(* IEC 61131-3 sources: cc_kush_rewrite/POUs, 10 files *)

(* ---- GLOBAL.st ---- *)
VAR_GLOBAL
	// Системные ФБ
	PULSE : BLINK;
	PULSE_RTRIG : R_TRIG;

	// Системные флаги
	xStateEmergencyStop : BOOL; // Система была аварийно остановлена
	xStateErrorAcceptIdle : BOOL; // Невозможно принять коэффицент шихтования по заданию оператора - сумма коэффицентов не равна 100
	xStateErrorCheckReady : BOOL; // Проверки стадии готовности к пуску провалились
	xStateAutoWorking : BOOL; // Система полностью запущена и работает в автоматическом режиме
	// Расчёт КИУМ
	ICUR_PRECENT : REAL; // Коэффициент использования установленной мощности (в процентах)
	rElectricityMeter : REAL; // Раход электроэнергии

	// Ограничение производительности
	EFFICIENCY_LIMIT_RATE : REAL := 1; // Коэффицент ограничения производительности (0-1)

	// Переменные симуляции
	SIMULATION : BOOL := FALSE;
	SIMULATION_BUNKER_WEIGHT : BOOL := FALSE; // Включение симуляции расхода и пополнения веса бункеров

	// == MODBUS РЕГИСТРЫ ДЛЯ SCADA ==
	// Массив регистров для передачи данных в SCADA систему
	awModbusInputRegisters : ARRAY [0..511] OF WORD; // Modbus Input регистры
	awModbusHoldingRegisters : ARRAY [0..511] OF WORD; // Modbus Holding регистры

	// == СИГНАЛЫ СВЯЗИ СО SCADA ==
	SCADA_HEARTBEAT : BOOL := FALSE; // Пульсирующий сигнал от SCADA (0 → 1 → 0) для контроля связи

END_VAR
VAR_GLOBAL RETAIN
	// == КРИТИЧЕСКИЕ НАСТРОЙКИ ==
	DISABLE_AUTO_STOPPING : BOOL := FALSE; // Отключение автоматических блокировок по цепям безопасности механизмов
	DISABLE_AUTO_STOPPING_DEPENDENCIES : BOOL := FALSE; 			// Отключение автоматических блокировок по блокировочным зависимостям
	DISABLE_AUTO_STOPPING_DEPENDENCIES_BUNKER1 : BOOL := FALSE; 	// Отключение автоматических блокировок бункера 1
	DISABLE_AUTO_STOPPING_DEPENDENCIES_BUNKER2 : BOOL := FALSE; 	// Отключение автоматических блокировок бункера 2
	DISABLE_AUTO_STOPPING_DEPENDENCIES_BUNKER3 : BOOL := FALSE; 	// Отключение автоматических блокировок бункера 3
	DISABLE_AUTO_STOPPING_DEPENDENCIES_CONVEYOR : BOOL := FALSE; 	// Отключение автоматических блокировок сборного конвейера
	DISABLE_AUTO_STOPPING_DEPENDENCIES_DUMPER : BOOL := FALSE; 		// Отключение автоматических блокировок отвалообразователя

	DISABLE_AUTO_STOPPING_SCADA_COMMUNICATION : BOOL := TRUE; // Отключение автоматических блокировок по потере связи со SCADA
	DISABLE_AUTO_STOPPING_CURRENT : BOOL := FALSE; // Отключение автоматических блокировок по значению тока
	BUNKER_INSTANT_STOP : BOOL := FALSE; // Флаг мгновенной остановки бункеров (TRUE = одновременная остановка всех 3-х бункеров, FALSE = последовательная остановка)

	// == УСТАВКИ ==
	VFD_FREQUENCY_MAX : REAL := 50;
	VFD_FREQUENCY_STEP : REAL := 2;
	VFD_FREQUENCY_INACCURANCY : REAL := 0.5;
	VFD_FREQUENCY_SYNC_TOLERANCE : REAL := 1.5; // Допустимая разница частот для синхронизации моторов

		// == ПАРАМЕТРЫ АЦП/ЦАП ДЛЯ ЧРП ==
	VFD_ADC_MAX : INT := 27648; // Максимальный код АЦП (аналоговый вход/выход)
	VFD_ADC_MIN : INT := 0; // Минимальный код АЦП
	VFD_FREQ_MIN : REAL := 0.0; // Минимальная частота ЧРП (Гц)
	VFD_FREQ_MAX_RANGE : REAL := 50.0; // Максимальная частота для масштабирования АЦП (Гц)

	// == ПАРАМЕТРЫ ТОКА 4-20 мА ==
	VFD_CURRENT_MIN : REAL := 4.0; // Минимальный ток (мА)
	VFD_CURRENT_MAX : REAL := 20.0; // Максимальный ток (мА)
	VFD_CURRENT_ALARM_LL : REAL := 3.8; // Аварийно низкий уровень тока (обрыв линии)
	VFD_CURRENT_ALARM_L : REAL := 4.5; // Низкий уровень тока
	VFD_CURRENT_ALARM_H : REAL := 19.5; // Высокий уровень тока
	VFD_CURRENT_ALARM_HH : REAL := 20.2; // Аварийно высокий уровень тока (перегрузка)

	// == ПАРАМЕТРЫ ДИАПАЗОНА ТЕМПЕРАТУР ==
	TEMP_BEARING_MIN : REAL := 0.0; // Минимальная температура подшипникового узла (°C)
	TEMP_BEARING_MAX : REAL := 100.0; // Максимальная температура подшипникового узла (°C)

	// Настройка виброобрушения
	VIBRATOR_SETTINGS : ST_BunkerVibratorSettings := (
		TIME_ACTIVE := T#15S,
		TIME_PAUSE_VIBRATOR := T#30S,
		TIME_PAUSE_FB := T#30S,
		COUNT_CYCLE := 3
		);

	// Настройка пневмообрушения
	PNEUMO_SETTINGS : ST_BunkerVibratorSettings := (
		TIME_ACTIVE := T#10S,
		TIME_PAUSE_VIBRATOR := T#10S,
		TIME_PAUSE_FB := T#30S,
		COUNT_CYCLE := 3
		);

	// Опция плавного задания частоты
	VFD_SMOOTH_SET_FREQUENCY : BOOL := FALSE;

	// Таймеры последовательного запуска механизмов в автоматическом режиме
	TIME_AFTER_START_DUMPER : TIME := T#120S; // Время ожидания после запуска отвалообразователя
	TIME_AFTER_START_CONVEYOR : TIME := T#120S; // Время ожидания после запуска конвейера
	TIME_AFTER_START_BUNKER_1 : TIME := T#120S; // Время ожидания после запуска бункера 1
	TIME_AFTER_START_BUNKER_2 : TIME := T#120S; // Время ожидания после запуска бункера 2
	TIME_AFTER_START_BUNKER_3 : TIME := T#120S; // Время ожидания после запуска бункера 3

	// Таймеры контроля выполнения команд (тайм-ауты)
	TIME_TIMEOUT_STOP_DUMPER : TIME := T#30S; // Тайм-аут остановки отвалообразователя (WORK → IDLE)
	TIME_TIMEOUT_STOP_CONVEYOR : TIME := T#30S; // Тайм-аут остановки конвейера (WORK → IDLE)
	TIME_TIMEOUT_ROTATION_DUMPER : TIME := T#20S; // Тайм-аут выполнения команд поворота дампера
	TIME_TIMEOUT_STOP_BUNKER : TIME := T#20S; // Тайм-аут остановки вибропитателей бункера (WORK → IDLE)

	// Таймер ожидания пропавшего сигнала обратной связи работы механизма
	TIME_WAITING_FEEDBACK : TIME := T#0S;

	// == ПАРАМЕТРЫ СВЯЗИ СО SCADA ==
	SCADA_HEARTBEAT_TIMEOUT : TIME := T#5S; // Таймаут отсутствия изменений heartbeat сигнала (потеря связи)

	// Таймаут контроля суммы пропорций в режиме WORK
	BUNKER_PROPORTION_SUM_TIMEOUT : TIME := T#20S; // Время ожидания корректировки суммы пропорций оператором (сумма должна быть = 100%)

	// Скорость конвейера
	CONVEYOR_DEAFULT_SPEED : REAL := -1;

	// Температура подшипникового узла мотора вибропитателя
	MOTOR_VIBFEEDER_TEMP_POINTS : ST_AlarmSetpoints := (
		LL_Value := -1,
		L_Value := -1,
		H_Value := -1,
		HH_Value := -1);
	// Ток мотора вибропитателя
	MOTOR_VIBFEEDER_CURRENT_POINTS : ST_AlarmSetpoints := (
		LL_Value := -1,
		L_Value := -1,
		H_Value := -1,
		HH_Value := -1);
	// Ток мотора вибратора
	MOTOR_VIBRATOR_CURRENT_POINTS : ST_AlarmSetpoints := (
		LL_Value := -1,
		L_Value := -1,
		H_Value := -1,
		HH_Value := -1);
	// Ток мотора конвейера отвалообразователя
	MOTOR_CONVEYOR_CURRENT_POINTS : ST_AlarmSetpoints := (
		LL_Value := -1,
		L_Value := -1,
		H_Value := -1,
		HH_Value := -1);
	// Ток мотора конвейера сборного
	MOTOR_CONVEYOR_PREFABRICATED_CURRENT_POINTS : ST_AlarmSetpoints := (
		LL_Value := -1,
		L_Value := -1,
		H_Value := -1,
		HH_Value := -1);
	// Ток мотора поворота отвалообразователя
	MOTOR_ROTATION_CURRENT_POINTS : ST_AlarmSetpoints := (
		LL_Value := -1,
		L_Value := -1,
		H_Value := -1,
		HH_Value := -1);

	// Предпусковая сигнализация конвейера отвалообразователя
	DUMPER_CONVEYOR_PRESTART_ALARM_SETTINGS : ST_PreStartAlarmSettings := (
		OPTION_ENABLE := TRUE, // Опция на включение ППЗ в алгоритм
		TIME_FIRST_SIGNAL := T#3S, // Время звучания первого сигнала
		TIME_FIRST_SIGNAL_PAUSE := T#3S, // Пауза после первого сигнала
		TIME_SECOND_SIGNAL := T#3S, // Время звучания второго сигнала
		TIME_SECOND_SIGNAL_PAUSE := T#3S); // Пауза после втотрого сигнала

	// Предпусковая сигнализация сборного конвейера
	CONVEYOR_PRESTART_ALARM_SETTINGS : ST_PreStartAlarmSettings := (
		OPTION_ENABLE := TRUE, // Опция на включение ППЗ в алгоритм
		TIME_FIRST_SIGNAL := T#3S, // Время звучания первого сигнала
		TIME_FIRST_SIGNAL_PAUSE := T#3S, // Пауза после первого сигнала
		TIME_SECOND_SIGNAL := T#3S, // Время звучания второго сигнала
		TIME_SECOND_SIGNAL_PAUSE := T#3S); // Пауза после втотрого сигнала

	// Световая индикация Гц
	ANNUNCIATOR_LIGHT_HZ : REAL := 2;

	// Частота мотора конвейера
	MOTOR_FREQUENCY_CONVEYOR : REAL := 50;
	// Частота мотора конвейера отвалообразователя
	MOTOR_FREQUENCY_DUMPER_CONVEYOR : REAL := 50;
	// Частота мотора поворота отвалообразователя
	MOTOR_FREQUENCY_DUMPER_ROTATION : REAL := -1;

	BUNKER_MINIMAL_WEIGHT :REAL := 0; // Уставка минимального веса бункера. Результат <= считывается алгоритмом как пустой бункер.

	// Уставки бункера
	PNEUMATIC_COLLAPSE_TIME : TIME := T#0S; // Уставка времени таймера пневмообрушения
	BUNKER_WORK_PRECENT_1 : REAL; // Уставка пропорции шихтования для бункера 1
	BUNKER_WORK_PRECENT_2 : REAL; // Уставка пропорции шихтования для бункера 2
	BUNKER_WORK_PRECENT_3 : REAL; // Уставка пропорции шихтования для бункера 3
	BUNKER_VIBFEEDER_START_FREQUENCY : REAL := 10.0; // Минимальная частота для запуска вибропитателей (Гц)
	BUNKER_VIBFEEDER_FREQUENCY_TARGET_SUM : REAL := 50.0; // Целевая суммарная частота вибропитателей (Гц)
    BUNKER_ENABLE_PID : BOOL := FALSE;
    BUNKER_ENABLE_PROPORTION_MONITORING : BOOL := FALSE;

	// == КОНТРОЛЬ МИНИМАЛЬНОЙ И МАКСИМАЛЬНОЙ ЧАСТОТЫ ВИБРОПИТАТЕЛЯ (ДЛЯ ПИД-РЕГУЛЯТОРА) ==
	BUNKER_VIBFEEDER_MIN_FREQUENCY_LIMIT : REAL := 5.0; // Минимальная допустимая частота вибропитателя (Гц) - при достижении этой уставки запускается таймер аварии
	BUNKER_VIBFEEDER_MIN_FREQUENCY_TIMEOUT : TIME := T#30S; // Время задержки перед аварийной остановкой при достижении минимальной частоты
	BUNKER_VIBFEEDER_MAX_FREQUENCY_LIMIT : REAL := 50.0; // Максимальная допустимая частота вибропитателя (Гц) - при достижении этой уставки запускается таймер аварии
	BUNKER_VIBFEEDER_MAX_FREQUENCY_TIMEOUT : TIME := T#30S; // Время задержки перед аварийной остановкой при достижении максимальной частоты

	// Ручное задание частоты на бункер (работает в ручном режиме управления)
	BUNKER_1_FREQ_VIBFEEDER : REAL := 30;
	BUNKER_1_FREQ_VIBRATOR : REAL := 30;
	BUNKER_2_FREQ_VIBFEEDER : REAL := 30;
	BUNKER_2_FREQ_VIBRATOR : REAL := 30;
	BUNKER_3_FREQ_VIBFEEDER : REAL := 30;
	BUNKER_3_FREQ_VIBRATOR : REAL := 30;

	// Светофор бункера
	BUNKER_WEIGHT_LIGHT_RED : REAL := 90; // Уставка веса бункера для красного светофора
	BUNKER_WEIGHT_LIGHT_YELLOW : REAL := 80; // Уставка веса бункера для жёлтого светофора
	BUNKER_WEIGHT_LIGHT_GREEN : REAL := 50; // Уставка веса бункера для зелёного светофора

	BUNKER_WEIGHT_LIGHT_RED_SPECIAL : REAL := 10; // Уставка веса бункера для красного светофора, когда сырье закончилось и требуется остановить подачу материала в остальные бункеры для будущего алгоритма опустошения

	// Константы
	AMOUNT_BUNKER_MOTOR_VIBFEEDER : INT := 2;
	AMOUNT_BUNKER_MOTOR_VIBRATOR : INT := 4;
END_VAR

(* ---- FC_ModbusToSCADA.st ---- *)
FUNCTION FC_ModbusToSCADA : BOOL
VAR_INPUT
    stBunker : REFERENCE TO ARRAY [1..3] OF ST_Bunker;
    stDumper : REFERENCE TO ST_DUMPER;
    stConveyor : REFERENCE TO ST_ConveyorPrefabricated;
    stCommonSignals : REFERENCE TO ST_CommonSignals;
	stCommands : REFERENCE TO ST_Commands;
	eBunkerStageToSCADA : REFERENCE TO ARRAY[1..3] OF E_ScadaStatesDevice;
	eConveyorStageToSCADA : REFERENCE TO E_ScadaStatesDevice; // Состояние для SCADA конвейера
	eDumperStageToSCADA : REFERENCE TO E_ScadaStatesDevice; // Состояние для SCADA отвалообразователя
	eSystemStageToSCADA : REFERENCE TO E_ScadaStatesDevice; // Общее состояние системы для SCADA
	fbScadaCommunication : REFERENCE TO FB_ScadaCommunication; // Функциональный блок контроля связи со SCADA

END_VAR
VAR
	rTempTime : REAL;
END_VAR

// ========================================
// MODBUS РЕГИСТРЫ
// ========================================

// === HOLDING РЕГИСТРЫ (SCADA → PLC) - Чтение уставок ===

// Общие системные переменные и уставки (0-29)
// Регистры 0-1: BOOL флаги команд
FC_ModbusReadBool(pRegisters := ADR(awModbusHoldingRegisters), iRegisterIndex := 0, iBitIndex := 0, xValue => stCommands.cmdStartCommon.ixSignal);
FC_ModbusReadBool(pRegisters := ADR(awModbusHoldingRegisters), iRegisterIndex := 0, iBitIndex := 1, xValue => stCommands.cmdStopCommon.ixSignal);
FC_ModbusReadBool(pRegisters := ADR(awModbusHoldingRegisters), iRegisterIndex := 0, iBitIndex := 2, xValue => stCommands.cmdEmergencyStopCommon.ixSignal);
FC_ModbusReadBool(pRegisters := ADR(awModbusHoldingRegisters), iRegisterIndex := 0, iBitIndex := 3, xValue => stCommands.cmdResetAll.ixSignal);
FC_ModbusReadBool(pRegisters := ADR(awModbusHoldingRegisters), iRegisterIndex := 0, iBitIndex := 4, xValue => SCADA_HEARTBEAT);
//FC_ModbusReadBool(pRegisters := ADR(awModbusHoldingRegisters), iRegisterIndex := 0, iBitIndex := 5, xValue => DISABLE_AUTO_STOPPING_SCADA_COMMUNICATION);
FC_ModbusReadBool(pRegisters := ADR(awModbusHoldingRegisters), iRegisterIndex := 0, iBitIndex := 8, xValue => stCommands.cmdSetToRepair);
FC_ModbusReadBool(pRegisters := ADR(awModbusHoldingRegisters), iRegisterIndex := 0, iBitIndex := 9, xValue => stCommands.cmdSetToManual);
FC_ModbusReadBool(pRegisters := ADR(awModbusHoldingRegisters), iRegisterIndex := 0, iBitIndex := 10, xValue => stCommands.cmdSetToAuto);

// Уставки ЧРП (30-59)
// Регистры 30-31: BOOL флаги ЧРП
FC_ModbusReadBool(pRegisters := ADR(awModbusHoldingRegisters), iRegisterIndex := 30, iBitIndex := 0, xValue => VFD_SMOOTH_SET_FREQUENCY);

FC_ModbusReadReal(pRegisters := ADR(awModbusHoldingRegisters), iRegisterIndex := 32, rValue => VFD_FREQUENCY_MAX);
FC_ModbusReadReal(pRegisters := ADR(awModbusHoldingRegisters), iRegisterIndex := 34, rValue => VFD_FREQUENCY_STEP);
FC_ModbusReadReal(pRegisters := ADR(awModbusHoldingRegisters), iRegisterIndex := 36, rValue => VFD_FREQUENCY_INACCURANCY);
FC_ModbusReadReal(pRegisters := ADR(awModbusHoldingRegisters), iRegisterIndex := 38, rValue => VFD_FREQUENCY_SYNC_TOLERANCE);
FC_ModbusReadReal(pRegisters := ADR(awModbusHoldingRegisters), iRegisterIndex := 40, rValue => MOTOR_FREQUENCY_CONVEYOR);
FC_ModbusReadReal(pRegisters := ADR(awModbusHoldingRegisters), iRegisterIndex := 42, rValue => MOTOR_FREQUENCY_DUMPER_CONVEYOR);
FC_ModbusReadReal(pRegisters := ADR(awModbusHoldingRegisters), iRegisterIndex := 44, rValue => MOTOR_FREQUENCY_DUMPER_ROTATION);
FC_ModbusReadReal(pRegisters := ADR(awModbusHoldingRegisters), iRegisterIndex := 46, rValue => CONVEYOR_DEAFULT_SPEED);

// Уставки бункеров (60-89)
// Регистры 60-61: BOOL флаги (резерв)
FC_ModbusReadReal(pRegisters := ADR(awModbusHoldingRegisters), iRegisterIndex := 62, rValue => BUNKER_WORK_PRECENT_1);
FC_ModbusReadReal(pRegisters := ADR(awModbusHoldingRegisters), iRegisterIndex := 64, rValue => BUNKER_WORK_PRECENT_2);
FC_ModbusReadReal(pRegisters := ADR(awModbusHoldingRegisters), iRegisterIndex := 66, rValue => BUNKER_WORK_PRECENT_3);
FC_ModbusReadReal(pRegisters := ADR(awModbusHoldingRegisters), iRegisterIndex := 68, rValue => BUNKER_MINIMAL_WEIGHT);
FC_ModbusReadReal(pRegisters := ADR(awModbusHoldingRegisters), iRegisterIndex := 70, rValue => BUNKER_WEIGHT_LIGHT_RED_SPECIAL);
FC_ModbusReadReal(pRegisters := ADR(awModbusHoldingRegisters), iRegisterIndex := 72, rValue => BUNKER_WEIGHT_LIGHT_RED);
FC_ModbusReadReal(pRegisters := ADR(awModbusHoldingRegisters), iRegisterIndex := 74, rValue => BUNKER_WEIGHT_LIGHT_YELLOW);
FC_ModbusReadReal(pRegisters := ADR(awModbusHoldingRegisters), iRegisterIndex := 76, rValue => BUNKER_WEIGHT_LIGHT_GREEN);

// Уставки аварийных значений - Температура (90-119)
// Регистры 90-91: BOOL флаги (резерв)
FC_ModbusReadReal(pRegisters := ADR(awModbusHoldingRegisters), iRegisterIndex := 92, rValue => MOTOR_VIBFEEDER_TEMP_POINTS.LL_Value);
FC_ModbusReadReal(pRegisters := ADR(awModbusHoldingRegisters), iRegisterIndex := 94, rValue => MOTOR_VIBFEEDER_TEMP_POINTS.L_Value);
FC_ModbusReadReal(pRegisters := ADR(awModbusHoldingRegisters), iRegisterIndex := 96, rValue => MOTOR_VIBFEEDER_TEMP_POINTS.H_Value);
FC_ModbusReadReal(pRegisters := ADR(awModbusHoldingRegisters), iRegisterIndex := 98, rValue => MOTOR_VIBFEEDER_TEMP_POINTS.HH_Value);

// Уставки аварийных значений - Ток (120-149)
// Регистры 120-121: BOOL флаги (резерв)
FC_ModbusReadReal(pRegisters := ADR(awModbusHoldingRegisters), iRegisterIndex := 122, rValue => MOTOR_VIBFEEDER_CURRENT_POINTS.LL_Value);
FC_ModbusReadReal(pRegisters := ADR(awModbusHoldingRegisters), iRegisterIndex := 124, rValue => MOTOR_VIBFEEDER_CURRENT_POINTS.L_Value);
FC_ModbusReadReal(pRegisters := ADR(awModbusHoldingRegisters), iRegisterIndex := 126, rValue => MOTOR_VIBFEEDER_CURRENT_POINTS.H_Value);
FC_ModbusReadReal(pRegisters := ADR(awModbusHoldingRegisters), iRegisterIndex := 128, rValue => MOTOR_VIBFEEDER_CURRENT_POINTS.HH_Value);
FC_ModbusReadReal(pRegisters := ADR(awModbusHoldingRegisters), iRegisterIndex := 130, rValue => MOTOR_VIBRATOR_CURRENT_POINTS.LL_Value);
FC_ModbusReadReal(pRegisters := ADR(awModbusHoldingRegisters), iRegisterIndex := 132, rValue => MOTOR_VIBRATOR_CURRENT_POINTS.L_Value);
FC_ModbusReadReal(pRegisters := ADR(awModbusHoldingRegisters), iRegisterIndex := 134, rValue => MOTOR_VIBRATOR_CURRENT_POINTS.H_Value);
FC_ModbusReadReal(pRegisters := ADR(awModbusHoldingRegisters), iRegisterIndex := 136, rValue => MOTOR_VIBRATOR_CURRENT_POINTS.HH_Value);
FC_ModbusReadReal(pRegisters := ADR(awModbusHoldingRegisters), iRegisterIndex := 138, rValue => MOTOR_CONVEYOR_CURRENT_POINTS.LL_Value);
FC_ModbusReadReal(pRegisters := ADR(awModbusHoldingRegisters), iRegisterIndex := 140, rValue => MOTOR_CONVEYOR_CURRENT_POINTS.L_Value);
FC_ModbusReadReal(pRegisters := ADR(awModbusHoldingRegisters), iRegisterIndex := 142, rValue => MOTOR_CONVEYOR_CURRENT_POINTS.H_Value);
FC_ModbusReadReal(pRegisters := ADR(awModbusHoldingRegisters), iRegisterIndex := 144, rValue => MOTOR_CONVEYOR_CURRENT_POINTS.HH_Value);
FC_ModbusReadReal(pRegisters := ADR(awModbusHoldingRegisters), iRegisterIndex := 146, rValue => MOTOR_ROTATION_CURRENT_POINTS.LL_Value);
FC_ModbusReadReal(pRegisters := ADR(awModbusHoldingRegisters), iRegisterIndex := 148, rValue => MOTOR_ROTATION_CURRENT_POINTS.L_Value);

// Уставки времени (150-179)
// Регистры 150-151: Уставки связи со SCADA
FC_ModbusReadReal(pRegisters := ADR(awModbusHoldingRegisters), iRegisterIndex := 150, rValue => rTempTime);
SCADA_HEARTBEAT_TIMEOUT := REAL_TO_TIME(rTempTime * 1000); // Таймаут потери связи (секунды)

FC_ModbusReadReal(pRegisters := ADR(awModbusHoldingRegisters), iRegisterIndex := 152, rValue => MOTOR_ROTATION_CURRENT_POINTS.H_Value);
FC_ModbusReadReal(pRegisters := ADR(awModbusHoldingRegisters), iRegisterIndex := 154, rValue => MOTOR_ROTATION_CURRENT_POINTS.HH_Value);
FC_ModbusReadReal(pRegisters := ADR(awModbusHoldingRegisters), iRegisterIndex := 156, rValue => rTempTime);
//VIBRATOR_SETTINGS.TIME_ACTIVE := REAL_TO_TIME(rTempTime * 1000);
FC_ModbusReadReal(pRegisters := ADR(awModbusHoldingRegisters), iRegisterIndex := 158, rValue => rTempTime);
//VIBRATOR_SETTINGS.TIME_PAUSE_VIBRATOR := REAL_TO_TIME(rTempTime * 1000);
FC_ModbusReadReal(pRegisters := ADR(awModbusHoldingRegisters), iRegisterIndex := 160, rValue => rTempTime);
VIBRATOR_SETTINGS.TIME_PAUSE_FB := REAL_TO_TIME(rTempTime * 1000);
FC_ModbusReadReal(pRegisters := ADR(awModbusHoldingRegisters), iRegisterIndex := 162, rValue => rTempTime);
PNEUMO_SETTINGS.TIME_ACTIVE := REAL_TO_TIME(rTempTime * 1000);
FC_ModbusReadReal(pRegisters := ADR(awModbusHoldingRegisters), iRegisterIndex := 164, rValue => rTempTime);
PNEUMO_SETTINGS.TIME_PAUSE_VIBRATOR := REAL_TO_TIME(rTempTime * 1000);
FC_ModbusReadReal(pRegisters := ADR(awModbusHoldingRegisters), iRegisterIndex := 166, rValue => rTempTime);
PNEUMO_SETTINGS.TIME_PAUSE_FB := REAL_TO_TIME(rTempTime * 1000);
FC_ModbusReadReal(pRegisters := ADR(awModbusHoldingRegisters), iRegisterIndex := 168, rValue => rTempTime);
TIME_WAITING_FEEDBACK := REAL_TO_TIME(rTempTime * 1000);
FC_ModbusReadReal(pRegisters := ADR(awModbusHoldingRegisters), iRegisterIndex := 170, rValue => rTempTime);
PNEUMATIC_COLLAPSE_TIME := REAL_TO_TIME(rTempTime * 1000);
FC_ModbusReadReal(pRegisters := ADR(awModbusHoldingRegisters), iRegisterIndex := 172, rValue => rTempTime);
DUMPER_CONVEYOR_PRESTART_ALARM_SETTINGS.TIME_FIRST_SIGNAL := REAL_TO_TIME(rTempTime * 1000);
FC_ModbusReadReal(pRegisters := ADR(awModbusHoldingRegisters), iRegisterIndex := 174, rValue => rTempTime);
DUMPER_CONVEYOR_PRESTART_ALARM_SETTINGS.TIME_FIRST_SIGNAL_PAUSE := REAL_TO_TIME(rTempTime * 1000);
FC_ModbusReadReal(pRegisters := ADR(awModbusHoldingRegisters), iRegisterIndex := 176, rValue => rTempTime);
DUMPER_CONVEYOR_PRESTART_ALARM_SETTINGS.TIME_SECOND_SIGNAL := REAL_TO_TIME(rTempTime * 1000);
FC_ModbusReadReal(pRegisters := ADR(awModbusHoldingRegisters), iRegisterIndex := 178, rValue => rTempTime);
DUMPER_CONVEYOR_PRESTART_ALARM_SETTINGS.TIME_SECOND_SIGNAL_PAUSE := REAL_TO_TIME(rTempTime * 1000);

// Уставки времени (продолжение) (180-209)
// Регистры 180-181: BOOL флаги (резерв)
FC_ModbusReadReal(pRegisters := ADR(awModbusHoldingRegisters), iRegisterIndex := 182, rValue => rTempTime);
CONVEYOR_PRESTART_ALARM_SETTINGS.TIME_FIRST_SIGNAL := REAL_TO_TIME(rTempTime * 1000);
FC_ModbusReadReal(pRegisters := ADR(awModbusHoldingRegisters), iRegisterIndex := 184, rValue => rTempTime);
CONVEYOR_PRESTART_ALARM_SETTINGS.TIME_FIRST_SIGNAL_PAUSE := REAL_TO_TIME(rTempTime * 1000);
FC_ModbusReadReal(pRegisters := ADR(awModbusHoldingRegisters), iRegisterIndex := 186, rValue => rTempTime);
CONVEYOR_PRESTART_ALARM_SETTINGS.TIME_SECOND_SIGNAL := REAL_TO_TIME(rTempTime * 1000);
FC_ModbusReadReal(pRegisters := ADR(awModbusHoldingRegisters), iRegisterIndex := 188, rValue => rTempTime);
CONVEYOR_PRESTART_ALARM_SETTINGS.TIME_SECOND_SIGNAL_PAUSE := REAL_TO_TIME(rTempTime * 1000);

// Команды - Отвалообразователь (210-239)
// Регистры 210-211: BOOL флаги управления отвалообразователем
FC_ModbusReadBool(pRegisters := ADR(awModbusHoldingRegisters), iRegisterIndex := 210, iBitIndex := 0, xValue => stDumper.cmdStartConveyor);
FC_ModbusReadBool(pRegisters := ADR(awModbusHoldingRegisters), iRegisterIndex := 210, iBitIndex := 1, xValue => stDumper.cmdStopConveyor);
FC_ModbusReadBool(pRegisters := ADR(awModbusHoldingRegisters), iRegisterIndex := 210, iBitIndex := 2, xValue => stDumper.cmdEmergencyStop);
FC_ModbusReadBool(pRegisters := ADR(awModbusHoldingRegisters), iRegisterIndex := 210, iBitIndex := 3, xValue => stDumper.cmdReset);
FC_ModbusReadBool(pRegisters := ADR(awModbusHoldingRegisters), iRegisterIndex := 210, iBitIndex := 8, xValue => stDumper.cmdSetModeRepair);
FC_ModbusReadBool(pRegisters := ADR(awModbusHoldingRegisters), iRegisterIndex := 210, iBitIndex := 9, xValue => stDumper.cmdSetModeManual);
FC_ModbusReadBool(pRegisters := ADR(awModbusHoldingRegisters), iRegisterIndex := 210, iBitIndex := 10, xValue => stDumper.cmdSetModeAuto);
FC_ModbusReadBool(pRegisters := ADR(awModbusHoldingRegisters), iRegisterIndex := 210, iBitIndex := 11, xValue => stDumper.cmdBuildCircuitOn);
FC_ModbusReadBool(pRegisters := ADR(awModbusHoldingRegisters), iRegisterIndex := 210, iBitIndex := 12, xValue => stDumper.cmdBuildCircuitOff);

FC_ModbusReadBool(pRegisters := ADR(awModbusHoldingRegisters), iRegisterIndex := 211, iBitIndex := 0, xValue => stDumper.cmdTurnLeft);
FC_ModbusReadBool(pRegisters := ADR(awModbusHoldingRegisters), iRegisterIndex := 211, iBitIndex := 1, xValue => stDumper.cmdTurnRight);
FC_ModbusReadBool(pRegisters := ADR(awModbusHoldingRegisters), iRegisterIndex := 211, iBitIndex := 2, xValue => stDumper.cmdStopRotation);
FC_ModbusReadBool(pRegisters := ADR(awModbusHoldingRegisters), iRegisterIndex := 211, iBitIndex := 11, xValue => stDumper.cmdBuildCircuitOnRotation);
FC_ModbusReadBool(pRegisters := ADR(awModbusHoldingRegisters), iRegisterIndex := 211, iBitIndex := 12, xValue => stDumper.cmdBuildCircuitOffRotation);

// Настройка - Отвалообразователь (210-239)
FC_ModbusReadBool(pRegisters := ADR(awModbusHoldingRegisters), iRegisterIndex := 212, iBitIndex := 0, xValue => DUMPER_CONVEYOR_PRESTART_ALARM_SETTINGS.OPTION_ENABLE);

// Команды - Конвейер (240-269)
// Регистры 240-241: BOOL флаги управления конвейером
FC_ModbusReadBool(pRegisters := ADR(awModbusHoldingRegisters), iRegisterIndex := 240, iBitIndex := 0, xValue => stConveyor.cmdStartConveyor);
FC_ModbusReadBool(pRegisters := ADR(awModbusHoldingRegisters), iRegisterIndex := 240, iBitIndex := 1, xValue => stConveyor.cmdStopConveyor);
FC_ModbusReadBool(pRegisters := ADR(awModbusHoldingRegisters), iRegisterIndex := 240, iBitIndex := 2, xValue => stConveyor.cmdEmergencyStop);
FC_ModbusReadBool(pRegisters := ADR(awModbusHoldingRegisters), iRegisterIndex := 240, iBitIndex := 3, xValue => stConveyor.cmdReset);
FC_ModbusReadBool(pRegisters := ADR(awModbusHoldingRegisters), iRegisterIndex := 240, iBitIndex := 8, xValue => stConveyor.cmdSetModeRepair);
FC_ModbusReadBool(pRegisters := ADR(awModbusHoldingRegisters), iRegisterIndex := 240, iBitIndex := 9, xValue => stConveyor.cmdSetModeManual);
FC_ModbusReadBool(pRegisters := ADR(awModbusHoldingRegisters), iRegisterIndex := 240, iBitIndex := 10, xValue => stConveyor.cmdSetModeAuto);
FC_ModbusReadBool(pRegisters := ADR(awModbusHoldingRegisters), iRegisterIndex := 240, iBitIndex := 11, xValue => stConveyor.cmdBuildCircuitOn);
FC_ModbusReadBool(pRegisters := ADR(awModbusHoldingRegisters), iRegisterIndex := 240, iBitIndex := 12, xValue => stConveyor.cmdBuildCircuitOff);

// Настройка - Конвейер (240-269)
FC_ModbusReadBool(pRegisters := ADR(awModbusHoldingRegisters), iRegisterIndex := 242, iBitIndex := 0, xValue => CONVEYOR_PRESTART_ALARM_SETTINGS.OPTION_ENABLE);

// Команды - Бункер 1 (270-299)
// Регистры 270-271: BOOL флаги управления бункером 1
FC_ModbusReadBool(pRegisters := ADR(awModbusHoldingRegisters), iRegisterIndex := 270, iBitIndex := 0, xValue => stBunker[1].cmdStartFeeder);
FC_ModbusReadBool(pRegisters := ADR(awModbusHoldingRegisters), iRegisterIndex := 270, iBitIndex := 1, xValue => stBunker[1].cmdStopFeeder);
FC_ModbusReadBool(pRegisters := ADR(awModbusHoldingRegisters), iRegisterIndex := 270, iBitIndex := 2, xValue => stBunker[1].cmdEmergencyStopVibFeeder);
FC_ModbusReadBool(pRegisters := ADR(awModbusHoldingRegisters), iRegisterIndex := 270, iBitIndex := 3, xValue => stBunker[1].cmdReset);
FC_ModbusReadBool(pRegisters := ADR(awModbusHoldingRegisters), iRegisterIndex := 270, iBitIndex := 8, xValue => stBunker[1].cmdSetModeRepair);
FC_ModbusReadBool(pRegisters := ADR(awModbusHoldingRegisters), iRegisterIndex := 270, iBitIndex := 9, xValue => stBunker[1].cmdSetModeManual);
FC_ModbusReadBool(pRegisters := ADR(awModbusHoldingRegisters), iRegisterIndex := 270, iBitIndex := 10, xValue => stBunker[1].cmdSetModeAuto);
FC_ModbusReadBool(pRegisters := ADR(awModbusHoldingRegisters), iRegisterIndex := 270, iBitIndex := 11, xValue => stBunker[1].cmdBuildCircuitOn);
FC_ModbusReadBool(pRegisters := ADR(awModbusHoldingRegisters), iRegisterIndex := 270, iBitIndex := 12, xValue => stBunker[1].cmdBuildCircuitOff);

FC_ModbusReadBool(pRegisters := ADR(awModbusHoldingRegisters), iRegisterIndex := 271, iBitIndex := 0, xValue => stBunker[1].cmdStartVibrator);
FC_ModbusReadBool(pRegisters := ADR(awModbusHoldingRegisters), iRegisterIndex := 271, iBitIndex := 1, xValue => stBunker[1].cmdStopVibrator);
FC_ModbusReadBool(pRegisters := ADR(awModbusHoldingRegisters), iRegisterIndex := 271, iBitIndex := 2, xValue => stBunker[1].cmdEmergencyStopVibrator);
FC_ModbusReadBool(pRegisters := ADR(awModbusHoldingRegisters), iRegisterIndex := 271, iBitIndex := 3, xValue => stBunker[1].cmdReset);
FC_ModbusReadBool(pRegisters := ADR(awModbusHoldingRegisters), iRegisterIndex := 271, iBitIndex := 4, xValue => stBunker[1].cmdAddVib1);
FC_ModbusReadBool(pRegisters := ADR(awModbusHoldingRegisters), iRegisterIndex := 271, iBitIndex := 5, xValue => stBunker[1].cmdAddVib2);
FC_ModbusReadBool(pRegisters := ADR(awModbusHoldingRegisters), iRegisterIndex := 271, iBitIndex := 6, xValue => stBunker[1].cmdAddVib3);
FC_ModbusReadBool(pRegisters := ADR(awModbusHoldingRegisters), iRegisterIndex := 271, iBitIndex := 7, xValue => stBunker[1].cmdAddVib4);
FC_ModbusReadBool(pRegisters := ADR(awModbusHoldingRegisters), iRegisterIndex := 271, iBitIndex := 8, xValue => stBunker[1].cmdVibratorSetModeRepair);
FC_ModbusReadBool(pRegisters := ADR(awModbusHoldingRegisters), iRegisterIndex := 271, iBitIndex := 9, xValue => stBunker[1].cmdVibratorSetModeManual);
FC_ModbusReadBool(pRegisters := ADR(awModbusHoldingRegisters), iRegisterIndex := 271, iBitIndex := 10, xValue => stBunker[1].cmdVibratorSetModeAuto);
FC_ModbusReadBool(pRegisters := ADR(awModbusHoldingRegisters), iRegisterIndex := 271, iBitIndex := 11, xValue => stBunker[1].cmdBuildCircuitOnVibrator);
FC_ModbusReadBool(pRegisters := ADR(awModbusHoldingRegisters), iRegisterIndex := 271, iBitIndex := 12, xValue => stBunker[1].cmdBuildCircuitOffVibrator);

FC_ModbusReadBool(pRegisters := ADR(awModbusHoldingRegisters), iRegisterIndex := 272, iBitIndex := 1, xValue => stBunker[1].cmdLighetSetColorRed);
FC_ModbusReadBool(pRegisters := ADR(awModbusHoldingRegisters), iRegisterIndex := 272, iBitIndex := 2, xValue => stBunker[1].cmdLighetSetColorYellow);
FC_ModbusReadBool(pRegisters := ADR(awModbusHoldingRegisters), iRegisterIndex := 272, iBitIndex := 3, xValue => stBunker[1].cmdLighetSetColorGreen);
FC_ModbusReadBool(pRegisters := ADR(awModbusHoldingRegisters), iRegisterIndex := 272, iBitIndex := 4, xValue => stBunker[1].cmdLighterSetModeAuto);
FC_ModbusReadBool(pRegisters := ADR(awModbusHoldingRegisters), iRegisterIndex := 272, iBitIndex := 8, xValue => stBunker[1].cmdLighterSetModeRepair);
FC_ModbusReadBool(pRegisters := ADR(awModbusHoldingRegisters), iRegisterIndex := 272, iBitIndex := 9, xValue => stBunker[1].cmdLighterSetModeManual);
FC_ModbusReadBool(pRegisters := ADR(awModbusHoldingRegisters), iRegisterIndex := 272, iBitIndex := 10, xValue => stBunker[1].cmdLighterSetModeAuto);

FC_ModbusReadReal(pRegisters := ADR(awModbusHoldingRegisters), iRegisterIndex := 278, rValue => BUNKER_1_FREQ_VIBRATOR);
FC_ModbusReadReal(pRegisters := ADR(awModbusHoldingRegisters), iRegisterIndex := 282, rValue => BUNKER_1_FREQ_VIBFEEDER);

// Команды - Бункер 2 (300-329)
// Регистры 300-301: BOOL флаги управления бункером 2
FC_ModbusReadBool(pRegisters := ADR(awModbusHoldingRegisters), iRegisterIndex := 300, iBitIndex := 0, xValue => stBunker[2].cmdStartFeeder);
FC_ModbusReadBool(pRegisters := ADR(awModbusHoldingRegisters), iRegisterIndex := 300, iBitIndex := 1, xValue => stBunker[2].cmdStopFeeder);
FC_ModbusReadBool(pRegisters := ADR(awModbusHoldingRegisters), iRegisterIndex := 300, iBitIndex := 2, xValue => stBunker[2].cmdEmergencyStopVibFeeder);
FC_ModbusReadBool(pRegisters := ADR(awModbusHoldingRegisters), iRegisterIndex := 300, iBitIndex := 3, xValue => stBunker[2].cmdReset);
FC_ModbusReadBool(pRegisters := ADR(awModbusHoldingRegisters), iRegisterIndex := 300, iBitIndex := 8, xValue => stBunker[2].cmdSetModeRepair);
FC_ModbusReadBool(pRegisters := ADR(awModbusHoldingRegisters), iRegisterIndex := 300, iBitIndex := 9, xValue => stBunker[2].cmdSetModeManual);
FC_ModbusReadBool(pRegisters := ADR(awModbusHoldingRegisters), iRegisterIndex := 300, iBitIndex := 10, xValue => stBunker[2].cmdSetModeAuto);
FC_ModbusReadBool(pRegisters := ADR(awModbusHoldingRegisters), iRegisterIndex := 300, iBitIndex := 11, xValue => stBunker[2].cmdBuildCircuitOn);
FC_ModbusReadBool(pRegisters := ADR(awModbusHoldingRegisters), iRegisterIndex := 300, iBitIndex := 12, xValue => stBunker[2].cmdBuildCircuitOff);

FC_ModbusReadBool(pRegisters := ADR(awModbusHoldingRegisters), iRegisterIndex := 301, iBitIndex := 0, xValue => stBunker[2].cmdStartVibrator);
FC_ModbusReadBool(pRegisters := ADR(awModbusHoldingRegisters), iRegisterIndex := 301, iBitIndex := 1, xValue => stBunker[2].cmdStopVibrator);
FC_ModbusReadBool(pRegisters := ADR(awModbusHoldingRegisters), iRegisterIndex := 301, iBitIndex := 2, xValue => stBunker[2].cmdEmergencyStopVibrator);
FC_ModbusReadBool(pRegisters := ADR(awModbusHoldingRegisters), iRegisterIndex := 301, iBitIndex := 3, xValue => stBunker[2].cmdReset);
FC_ModbusReadBool(pRegisters := ADR(awModbusHoldingRegisters), iRegisterIndex := 301, iBitIndex := 4, xValue => stBunker[2].cmdAddVib1);
FC_ModbusReadBool(pRegisters := ADR(awModbusHoldingRegisters), iRegisterIndex := 301, iBitIndex := 5, xValue => stBunker[2].cmdAddVib2);
FC_ModbusReadBool(pRegisters := ADR(awModbusHoldingRegisters), iRegisterIndex := 301, iBitIndex := 6, xValue => stBunker[2].cmdAddVib3);
FC_ModbusReadBool(pRegisters := ADR(awModbusHoldingRegisters), iRegisterIndex := 301, iBitIndex := 7, xValue => stBunker[2].cmdAddVib4);
FC_ModbusReadBool(pRegisters := ADR(awModbusHoldingRegisters), iRegisterIndex := 301, iBitIndex := 8, xValue => stBunker[2].cmdVibratorSetModeRepair);
FC_ModbusReadBool(pRegisters := ADR(awModbusHoldingRegisters), iRegisterIndex := 301, iBitIndex := 9, xValue => stBunker[2].cmdVibratorSetModeManual);
FC_ModbusReadBool(pRegisters := ADR(awModbusHoldingRegisters), iRegisterIndex := 301, iBitIndex := 10, xValue => stBunker[2].cmdVibratorSetModeAuto);
FC_ModbusReadBool(pRegisters := ADR(awModbusHoldingRegisters), iRegisterIndex := 301, iBitIndex := 11, xValue => stBunker[2].cmdBuildCircuitOnVibrator);
FC_ModbusReadBool(pRegisters := ADR(awModbusHoldingRegisters), iRegisterIndex := 301, iBitIndex := 12, xValue => stBunker[2].cmdBuildCircuitOffVibrator);

FC_ModbusReadBool(pRegisters := ADR(awModbusHoldingRegisters), iRegisterIndex := 302, iBitIndex := 1, xValue => stBunker[2].cmdLighetSetColorRed);
FC_ModbusReadBool(pRegisters := ADR(awModbusHoldingRegisters), iRegisterIndex := 302, iBitIndex := 2, xValue => stBunker[2].cmdLighetSetColorYellow);
FC_ModbusReadBool(pRegisters := ADR(awModbusHoldingRegisters), iRegisterIndex := 302, iBitIndex := 3, xValue => stBunker[2].cmdLighetSetColorGreen);
FC_ModbusReadBool(pRegisters := ADR(awModbusHoldingRegisters), iRegisterIndex := 302, iBitIndex := 8, xValue => stBunker[2].cmdLighterSetModeRepair);
FC_ModbusReadBool(pRegisters := ADR(awModbusHoldingRegisters), iRegisterIndex := 302, iBitIndex := 9, xValue => stBunker[2].cmdLighterSetModeManual);
FC_ModbusReadBool(pRegisters := ADR(awModbusHoldingRegisters), iRegisterIndex := 302, iBitIndex := 10, xValue => stBunker[2].cmdLighterSetModeAuto);

FC_ModbusReadReal(pRegisters := ADR(awModbusHoldingRegisters), iRegisterIndex := 308, rValue => BUNKER_2_FREQ_VIBRATOR);
FC_ModbusReadReal(pRegisters := ADR(awModbusHoldingRegisters), iRegisterIndex := 312, rValue => BUNKER_2_FREQ_VIBFEEDER);

// Команды - Бункер 3 (330-359)
// Регистры 330-331: BOOL флаги управления бункером 3
FC_ModbusReadBool(pRegisters := ADR(awModbusHoldingRegisters), iRegisterIndex := 330, iBitIndex := 0, xValue => stBunker[3].cmdStartFeeder);
FC_ModbusReadBool(pRegisters := ADR(awModbusHoldingRegisters), iRegisterIndex := 330, iBitIndex := 1, xValue => stBunker[3].cmdStopFeeder);
FC_ModbusReadBool(pRegisters := ADR(awModbusHoldingRegisters), iRegisterIndex := 330, iBitIndex := 2, xValue => stBunker[3].cmdEmergencyStopVibFeeder);
FC_ModbusReadBool(pRegisters := ADR(awModbusHoldingRegisters), iRegisterIndex := 330, iBitIndex := 3, xValue => stBunker[3].cmdReset);
FC_ModbusReadBool(pRegisters := ADR(awModbusHoldingRegisters), iRegisterIndex := 330, iBitIndex := 8, xValue => stBunker[3].cmdSetModeRepair);
FC_ModbusReadBool(pRegisters := ADR(awModbusHoldingRegisters), iRegisterIndex := 330, iBitIndex := 9, xValue => stBunker[3].cmdSetModeManual);
FC_ModbusReadBool(pRegisters := ADR(awModbusHoldingRegisters), iRegisterIndex := 330, iBitIndex := 10, xValue => stBunker[3].cmdSetModeAuto);
FC_ModbusReadBool(pRegisters := ADR(awModbusHoldingRegisters), iRegisterIndex := 330, iBitIndex := 11, xValue => stBunker[3].cmdBuildCircuitOn);
FC_ModbusReadBool(pRegisters := ADR(awModbusHoldingRegisters), iRegisterIndex := 330, iBitIndex := 12, xValue => stBunker[3].cmdBuildCircuitOff);

FC_ModbusReadBool(pRegisters := ADR(awModbusHoldingRegisters), iRegisterIndex := 331, iBitIndex := 0, xValue => stBunker[3].cmdStartVibrator);
FC_ModbusReadBool(pRegisters := ADR(awModbusHoldingRegisters), iRegisterIndex := 331, iBitIndex := 1, xValue => stBunker[3].cmdStopVibrator);
FC_ModbusReadBool(pRegisters := ADR(awModbusHoldingRegisters), iRegisterIndex := 331, iBitIndex := 2, xValue => stBunker[3].cmdEmergencyStopVibrator);
FC_ModbusReadBool(pRegisters := ADR(awModbusHoldingRegisters), iRegisterIndex := 331, iBitIndex := 3, xValue => stBunker[3].cmdReset);
FC_ModbusReadBool(pRegisters := ADR(awModbusHoldingRegisters), iRegisterIndex := 331, iBitIndex := 4, xValue => stBunker[3].cmdAddVib1);
FC_ModbusReadBool(pRegisters := ADR(awModbusHoldingRegisters), iRegisterIndex := 331, iBitIndex := 5, xValue => stBunker[3].cmdAddVib2);
FC_ModbusReadBool(pRegisters := ADR(awModbusHoldingRegisters), iRegisterIndex := 331, iBitIndex := 6, xValue => stBunker[3].cmdAddVib3);
FC_ModbusReadBool(pRegisters := ADR(awModbusHoldingRegisters), iRegisterIndex := 331, iBitIndex := 7, xValue => stBunker[3].cmdAddVib4);
FC_ModbusReadBool(pRegisters := ADR(awModbusHoldingRegisters), iRegisterIndex := 331, iBitIndex := 8, xValue => stBunker[3].cmdVibratorSetModeRepair);
FC_ModbusReadBool(pRegisters := ADR(awModbusHoldingRegisters), iRegisterIndex := 331, iBitIndex := 9, xValue => stBunker[3].cmdVibratorSetModeManual);
FC_ModbusReadBool(pRegisters := ADR(awModbusHoldingRegisters), iRegisterIndex := 331, iBitIndex := 10, xValue => stBunker[3].cmdVibratorSetModeAuto);
FC_ModbusReadBool(pRegisters := ADR(awModbusHoldingRegisters), iRegisterIndex := 331, iBitIndex := 11, xValue => stBunker[3].cmdBuildCircuitOnVibrator);
FC_ModbusReadBool(pRegisters := ADR(awModbusHoldingRegisters), iRegisterIndex := 331, iBitIndex := 12, xValue => stBunker[3].cmdBuildCircuitOffVibrator);

FC_ModbusReadBool(pRegisters := ADR(awModbusHoldingRegisters), iRegisterIndex := 332, iBitIndex := 1, xValue => stBunker[3].cmdLighetSetColorRed);
FC_ModbusReadBool(pRegisters := ADR(awModbusHoldingRegisters), iRegisterIndex := 332, iBitIndex := 2, xValue => stBunker[3].cmdLighetSetColorYellow);
FC_ModbusReadBool(pRegisters := ADR(awModbusHoldingRegisters), iRegisterIndex := 332, iBitIndex := 3, xValue => stBunker[3].cmdLighetSetColorGreen);
FC_ModbusReadBool(pRegisters := ADR(awModbusHoldingRegisters), iRegisterIndex := 332, iBitIndex := 8, xValue => stBunker[3].cmdLighterSetModeRepair);
FC_ModbusReadBool(pRegisters := ADR(awModbusHoldingRegisters), iRegisterIndex := 332, iBitIndex := 9, xValue => stBunker[3].cmdLighterSetModeManual);
FC_ModbusReadBool(pRegisters := ADR(awModbusHoldingRegisters), iRegisterIndex := 332, iBitIndex := 10, xValue => stBunker[3].cmdLighterSetModeAuto);

FC_ModbusReadReal(pRegisters := ADR(awModbusHoldingRegisters), iRegisterIndex := 338, rValue => BUNKER_3_FREQ_VIBRATOR);
FC_ModbusReadReal(pRegisters := ADR(awModbusHoldingRegisters), iRegisterIndex := 342, rValue => BUNKER_3_FREQ_VIBFEEDER);

// === INPUT РЕГИСТРЫ (PLC → SCADA) - Запись данных мониторинга ===

// Общие системные статусы (0-29)
// Регистры 0-1: BOOL флаги статусов системы
FC_ModbusWriteBool(pRegisters := ADR(awModbusInputRegisters), iRegisterIndex := 0, iBitIndex := 0, xValue := xStateAutoWorking);
FC_ModbusWriteBool(pRegisters := ADR(awModbusInputRegisters), iRegisterIndex := 0, iBitIndex := 1, xValue := xStateEmergencyStop);
FC_ModbusWriteBool(pRegisters := ADR(awModbusInputRegisters), iRegisterIndex := 0, iBitIndex := 2, xValue := xStateErrorCheckReady);
FC_ModbusWriteBool(pRegisters := ADR(awModbusInputRegisters), iRegisterIndex := 0, iBitIndex := 3, xValue := xStateErrorAcceptIdle);
FC_ModbusWriteBool(pRegisters := ADR(awModbusInputRegisters), iRegisterIndex := 0, iBitIndex := 4, xValue := fbScadaCommunication.qxCommunicationOk);
FC_ModbusWriteBool(pRegisters := ADR(awModbusInputRegisters), iRegisterIndex := 0, iBitIndex := 5, xValue := fbScadaCommunication.qxCommunicationLost);
FC_ModbusWriteBool(pRegisters := ADR(awModbusInputRegisters), iRegisterIndex := 0, iBitIndex := 6, xValue := fbScadaCommunication.qxSignalChanged);
FC_ModbusWriteBool(pRegisters := ADR(awModbusInputRegisters), iRegisterIndex := 0, iBitIndex := 7, xValue := stCommonSignals.fbQF1.qxSignal);
FC_ModbusWriteBool(pRegisters := ADR(awModbusInputRegisters), iRegisterIndex := 0, iBitIndex := 12, xValue := (stBunker[1].xStateRemoteAuto AND stBunker[2].xStateRemoteAuto AND stBunker[3].xStateRemoteAuto AND stDumper.xStateRemoteAuto AND stConveyor.xStateRemoteAuto));
FC_ModbusWriteBool(pRegisters := ADR(awModbusInputRegisters), iRegisterIndex := 0, iBitIndex := 13, xValue := NOT(stBunker[1].xStateRemoteAuto AND stBunker[2].xStateRemoteAuto AND stBunker[3].xStateRemoteAuto AND stDumper.xStateRemoteAuto AND stConveyor.xStateRemoteAuto));

FC_ModbusWriteBool(pRegisters := ADR(awModbusInputRegisters), iRegisterIndex := 0, iBitIndex := 15, xValue := SIMULATION);

FC_ModbusWriteReal(pRegisters := ADR(awModbusInputRegisters), iRegisterIndex := 2, rValue := ICUR_PRECENT);

// Регистр 4: Общее состояние системы для SCADA
FC_ModbusWriteInt(pRegisters := ADR(awModbusInputRegisters), iRegisterIndex := 4, iValue := eSystemStageToSCADA);

// Бункер 1 (30-89)
// Регистры 30-31: BOOL флаги статусов бункера 1
FC_ModbusWriteBool(pRegisters := ADR(awModbusInputRegisters), iRegisterIndex := 30, iBitIndex := 0, xValue := stBunker[1].xStateWarning);
FC_ModbusWriteBool(pRegisters := ADR(awModbusInputRegisters), iRegisterIndex := 30, iBitIndex := 1, xValue := stBunker[1].xStateFailure);
FC_ModbusWriteBool(pRegisters := ADR(awModbusInputRegisters), iRegisterIndex := 30, iBitIndex := 12, xValue := stBunker[1].xStateRemoteAuto);
FC_ModbusWriteBool(pRegisters := ADR(awModbusInputRegisters), iRegisterIndex := 30, iBitIndex := 13, xValue := stBunker[1].xStateRemoteManual);
FC_ModbusWriteBool(pRegisters := ADR(awModbusInputRegisters), iRegisterIndex := 30, iBitIndex := 14, xValue := stBunker[1].xStateRemoteRepair);

// Регистр 31: состояния режима управления светофора и вибраторов
FC_ModbusWriteBool(pRegisters := ADR(awModbusInputRegisters), iRegisterIndex := 31, iBitIndex := 9, xValue := stBunker[1].xLighterStateRemoteAuto);
FC_ModbusWriteBool(pRegisters := ADR(awModbusInputRegisters), iRegisterIndex := 31, iBitIndex := 10, xValue := stBunker[1].xLighterStateRemoteManual);
FC_ModbusWriteBool(pRegisters := ADR(awModbusInputRegisters), iRegisterIndex := 31, iBitIndex := 11, xValue := stBunker[1].xLighterStateRemoteRepair);
FC_ModbusWriteBool(pRegisters := ADR(awModbusInputRegisters), iRegisterIndex := 31, iBitIndex := 12, xValue := stBunker[1].xVibratorStateRemoteAuto);
FC_ModbusWriteBool(pRegisters := ADR(awModbusInputRegisters), iRegisterIndex := 31, iBitIndex := 13, xValue := stBunker[1].xVibratorStateRemoteManual);
FC_ModbusWriteBool(pRegisters := ADR(awModbusInputRegisters), iRegisterIndex := 31, iBitIndex := 14, xValue := stBunker[1].xVibratorStateRemoteRepair);

FC_ModbusWriteReal(pRegisters := ADR(awModbusInputRegisters), iRegisterIndex := 32, rValue := stBunker[1].rWeight);
FC_ModbusWriteReal(pRegisters := ADR(awModbusInputRegisters), iRegisterIndex := 34, rValue := stBunker[1].rProportionActual);
FC_ModbusWriteReal(pRegisters := ADR(awModbusInputRegisters), iRegisterIndex := 38, rValue := stBunker[1].cmdDumpingPrecent);
FC_ModbusWriteReal(pRegisters := ADR(awModbusInputRegisters), iRegisterIndex := 40, rValue := stBunker[1].MotorVibrator[1].VFD.qrOutFrequency);
FC_ModbusWriteReal(pRegisters := ADR(awModbusInputRegisters), iRegisterIndex := 42, rValue := stBunker[1].MotorVibrator[1].VFD.rActualFrequency);
FC_ModbusWriteReal(pRegisters := ADR(awModbusInputRegisters), iRegisterIndex := 44, rValue := stBunker[1].MotorVibrator[1].VFD.wMotorCurrent.rTag);
FC_ModbusWriteReal(pRegisters := ADR(awModbusInputRegisters), iRegisterIndex := 46, rValue := stBunker[1].MotorVibrator[2].VFD.qrOutFrequency);
FC_ModbusWriteReal(pRegisters := ADR(awModbusInputRegisters), iRegisterIndex := 48, rValue := stBunker[1].MotorVibrator[2].VFD.rActualFrequency);
FC_ModbusWriteReal(pRegisters := ADR(awModbusInputRegisters), iRegisterIndex := 50, rValue := stBunker[1].MotorVibrator[2].VFD.wMotorCurrent.rTag);
FC_ModbusWriteReal(pRegisters := ADR(awModbusInputRegisters), iRegisterIndex := 52, rValue := stBunker[1].MotorVibrator[3].VFD.qrOutFrequency);
FC_ModbusWriteReal(pRegisters := ADR(awModbusInputRegisters), iRegisterIndex := 54, rValue := stBunker[1].MotorVibrator[3].VFD.rActualFrequency);
FC_ModbusWriteReal(pRegisters := ADR(awModbusInputRegisters), iRegisterIndex := 56, rValue := stBunker[1].MotorVibrator[3].VFD.wMotorCurrent.rTag);
FC_ModbusWriteReal(pRegisters := ADR(awModbusInputRegisters), iRegisterIndex := 58, rValue := stBunker[1].MotorVibrator[4].VFD.qrOutFrequency);
FC_ModbusWriteReal(pRegisters := ADR(awModbusInputRegisters), iRegisterIndex := 60, rValue := stBunker[1].MotorVibrator[4].VFD.rActualFrequency);
FC_ModbusWriteReal(pRegisters := ADR(awModbusInputRegisters), iRegisterIndex := 62, rValue := stBunker[1].MotorVibrator[4].VFD.wMotorCurrent.rTag);
FC_ModbusWriteReal(pRegisters := ADR(awModbusInputRegisters), iRegisterIndex := 64, rValue := stBunker[1].MotorVibFeeder[1].VFD.qrOutFrequency);
FC_ModbusWriteReal(pRegisters := ADR(awModbusInputRegisters), iRegisterIndex := 66, rValue := stBunker[1].MotorVibFeeder[1].VFD.rActualFrequency);
FC_ModbusWriteReal(pRegisters := ADR(awModbusInputRegisters), iRegisterIndex := 68, rValue := stBunker[1].MotorVibFeeder[1].VFD.wMotorCurrent.rTag);
FC_ModbusWriteReal(pRegisters := ADR(awModbusInputRegisters), iRegisterIndex := 70, rValue := stBunker[1].MotorVibFeeder[2].VFD.qrOutFrequency);
FC_ModbusWriteReal(pRegisters := ADR(awModbusInputRegisters), iRegisterIndex := 72, rValue := stBunker[1].MotorVibFeeder[2].VFD.rActualFrequency);
FC_ModbusWriteReal(pRegisters := ADR(awModbusInputRegisters), iRegisterIndex := 74, rValue := stBunker[1].MotorVibFeeder[2].VFD.wMotorCurrent.rTag);
FC_ModbusWriteReal(pRegisters := ADR(awModbusInputRegisters), iRegisterIndex := 76, rValue := stBunker[1].MotorVibFeeder[1].rTempBearing[1]);
FC_ModbusWriteReal(pRegisters := ADR(awModbusInputRegisters), iRegisterIndex := 78, rValue := stBunker[1].MotorVibFeeder[1].rTempBearing[2]);
FC_ModbusWriteReal(pRegisters := ADR(awModbusInputRegisters), iRegisterIndex := 80, rValue := stBunker[1].MotorVibFeeder[2].rTempBearing[1]);
FC_ModbusWriteReal(pRegisters := ADR(awModbusInputRegisters), iRegisterIndex := 82, rValue := stBunker[1].MotorVibFeeder[2].rTempBearing[2]);

FC_ModbusWriteUInt(pRegisters := ADR(awModbusInputRegisters), iRegisterIndex := 84, uValue := eBunkerStageToSCADA[1]);

// Бункер 2 (90-149)
// Регистры 90-91: BOOL флаги статусов бункера 2
FC_ModbusWriteBool(pRegisters := ADR(awModbusInputRegisters), iRegisterIndex := 90, iBitIndex := 0, xValue := stBunker[2].xStateWarning);
FC_ModbusWriteBool(pRegisters := ADR(awModbusInputRegisters), iRegisterIndex := 90, iBitIndex := 1, xValue := stBunker[2].xStateFailure);
FC_ModbusWriteBool(pRegisters := ADR(awModbusInputRegisters), iRegisterIndex := 90, iBitIndex := 12, xValue := stBunker[2].xStateRemoteAuto);
FC_ModbusWriteBool(pRegisters := ADR(awModbusInputRegisters), iRegisterIndex := 90, iBitIndex := 13, xValue := stBunker[2].xStateRemoteManual);
FC_ModbusWriteBool(pRegisters := ADR(awModbusInputRegisters), iRegisterIndex := 90, iBitIndex := 14, xValue := stBunker[2].xStateRemoteRepair);

// Регистр 91: состояния режима управления светофора и вибраторов
FC_ModbusWriteBool(pRegisters := ADR(awModbusInputRegisters), iRegisterIndex := 91, iBitIndex := 9, xValue := stBunker[2].xLighterStateRemoteAuto);
FC_ModbusWriteBool(pRegisters := ADR(awModbusInputRegisters), iRegisterIndex := 91, iBitIndex := 10, xValue := stBunker[2].xLighterStateRemoteManual);
FC_ModbusWriteBool(pRegisters := ADR(awModbusInputRegisters), iRegisterIndex := 91, iBitIndex := 11, xValue := stBunker[2].xLighterStateRemoteRepair);
FC_ModbusWriteBool(pRegisters := ADR(awModbusInputRegisters), iRegisterIndex := 91, iBitIndex := 12, xValue := stBunker[2].xVibratorStateRemoteAuto);
FC_ModbusWriteBool(pRegisters := ADR(awModbusInputRegisters), iRegisterIndex := 91, iBitIndex := 13, xValue := stBunker[2].xVibratorStateRemoteManual);
FC_ModbusWriteBool(pRegisters := ADR(awModbusInputRegisters), iRegisterIndex := 91, iBitIndex := 14, xValue := stBunker[2].xVibratorStateRemoteRepair);

FC_ModbusWriteReal(pRegisters := ADR(awModbusInputRegisters), iRegisterIndex := 92, rValue := stBunker[2].rWeight);
FC_ModbusWriteReal(pRegisters := ADR(awModbusInputRegisters), iRegisterIndex := 94, rValue := stBunker[2].rProportionActual);
FC_ModbusWriteReal(pRegisters := ADR(awModbusInputRegisters), iRegisterIndex := 98, rValue := stBunker[2].cmdDumpingPrecent);
FC_ModbusWriteReal(pRegisters := ADR(awModbusInputRegisters), iRegisterIndex := 100, rValue := stBunker[2].MotorVibrator[1].VFD.qrOutFrequency);
FC_ModbusWriteReal(pRegisters := ADR(awModbusInputRegisters), iRegisterIndex := 102, rValue := stBunker[2].MotorVibrator[1].VFD.rActualFrequency);
FC_ModbusWriteReal(pRegisters := ADR(awModbusInputRegisters), iRegisterIndex := 104, rValue := stBunker[2].MotorVibrator[1].VFD.wMotorCurrent.rTag);
FC_ModbusWriteReal(pRegisters := ADR(awModbusInputRegisters), iRegisterIndex := 106, rValue := stBunker[2].MotorVibrator[2].VFD.qrOutFrequency);
FC_ModbusWriteReal(pRegisters := ADR(awModbusInputRegisters), iRegisterIndex := 108, rValue := stBunker[2].MotorVibrator[2].VFD.rActualFrequency);
FC_ModbusWriteReal(pRegisters := ADR(awModbusInputRegisters), iRegisterIndex := 110, rValue := stBunker[2].MotorVibrator[2].VFD.wMotorCurrent.rTag);
FC_ModbusWriteReal(pRegisters := ADR(awModbusInputRegisters), iRegisterIndex := 112, rValue := stBunker[2].MotorVibrator[3].VFD.qrOutFrequency);
FC_ModbusWriteReal(pRegisters := ADR(awModbusInputRegisters), iRegisterIndex := 114, rValue := stBunker[2].MotorVibrator[3].VFD.rActualFrequency);
FC_ModbusWriteReal(pRegisters := ADR(awModbusInputRegisters), iRegisterIndex := 116, rValue := stBunker[2].MotorVibrator[3].VFD.wMotorCurrent.rTag);
FC_ModbusWriteReal(pRegisters := ADR(awModbusInputRegisters), iRegisterIndex := 118, rValue := stBunker[2].MotorVibrator[4].VFD.qrOutFrequency);
FC_ModbusWriteReal(pRegisters := ADR(awModbusInputRegisters), iRegisterIndex := 120, rValue := stBunker[2].MotorVibrator[4].VFD.rActualFrequency);
FC_ModbusWriteReal(pRegisters := ADR(awModbusInputRegisters), iRegisterIndex := 122, rValue := stBunker[2].MotorVibrator[4].VFD.wMotorCurrent.rTag);
FC_ModbusWriteReal(pRegisters := ADR(awModbusInputRegisters), iRegisterIndex := 124, rValue := stBunker[2].MotorVibFeeder[1].VFD.qrOutFrequency);
FC_ModbusWriteReal(pRegisters := ADR(awModbusInputRegisters), iRegisterIndex := 126, rValue := stBunker[2].MotorVibFeeder[1].VFD.rActualFrequency);
FC_ModbusWriteReal(pRegisters := ADR(awModbusInputRegisters), iRegisterIndex := 128, rValue := stBunker[2].MotorVibFeeder[1].VFD.wMotorCurrent.rTag);
FC_ModbusWriteReal(pRegisters := ADR(awModbusInputRegisters), iRegisterIndex := 130, rValue := stBunker[2].MotorVibFeeder[2].VFD.qrOutFrequency);
FC_ModbusWriteReal(pRegisters := ADR(awModbusInputRegisters), iRegisterIndex := 132, rValue := stBunker[2].MotorVibFeeder[2].VFD.rActualFrequency);
FC_ModbusWriteReal(pRegisters := ADR(awModbusInputRegisters), iRegisterIndex := 134, rValue := stBunker[2].MotorVibFeeder[2].VFD.wMotorCurrent.rTag);
FC_ModbusWriteReal(pRegisters := ADR(awModbusInputRegisters), iRegisterIndex := 136, rValue := stBunker[2].MotorVibFeeder[1].rTempBearing[1]);
FC_ModbusWriteReal(pRegisters := ADR(awModbusInputRegisters), iRegisterIndex := 138, rValue := stBunker[2].MotorVibFeeder[1].rTempBearing[2]);
FC_ModbusWriteReal(pRegisters := ADR(awModbusInputRegisters), iRegisterIndex := 140, rValue := stBunker[2].MotorVibFeeder[2].rTempBearing[1]);
FC_ModbusWriteReal(pRegisters := ADR(awModbusInputRegisters), iRegisterIndex := 142, rValue := stBunker[2].MotorVibFeeder[2].rTempBearing[2]);

FC_ModbusWriteUInt(pRegisters := ADR(awModbusInputRegisters), iRegisterIndex := 144, uValue := eBunkerStageToSCADA[2]);

// Бункер 3 (150-209)
// Регистры 150-151: BOOL флаги статусов бункера 3
FC_ModbusWriteBool(pRegisters := ADR(awModbusInputRegisters), iRegisterIndex := 150, iBitIndex := 0, xValue := stBunker[3].xStateWarning);
FC_ModbusWriteBool(pRegisters := ADR(awModbusInputRegisters), iRegisterIndex := 150, iBitIndex := 1, xValue := stBunker[3].xStateFailure);
FC_ModbusWriteBool(pRegisters := ADR(awModbusInputRegisters), iRegisterIndex := 150, iBitIndex := 12, xValue := stBunker[3].xStateRemoteAuto);
FC_ModbusWriteBool(pRegisters := ADR(awModbusInputRegisters), iRegisterIndex := 150, iBitIndex := 13, xValue := stBunker[3].xStateRemoteManual);
FC_ModbusWriteBool(pRegisters := ADR(awModbusInputRegisters), iRegisterIndex := 150, iBitIndex := 14, xValue := stBunker[3].xStateRemoteRepair);

// Регистр 151: состояния режима управления светофора и вибраторов
FC_ModbusWriteBool(pRegisters := ADR(awModbusInputRegisters), iRegisterIndex := 151, iBitIndex := 9, xValue := stBunker[3].xLighterStateRemoteAuto);
FC_ModbusWriteBool(pRegisters := ADR(awModbusInputRegisters), iRegisterIndex := 151, iBitIndex := 10, xValue := stBunker[3].xLighterStateRemoteManual);
FC_ModbusWriteBool(pRegisters := ADR(awModbusInputRegisters), iRegisterIndex := 151, iBitIndex := 11, xValue := stBunker[3].xLighterStateRemoteRepair);
FC_ModbusWriteBool(pRegisters := ADR(awModbusInputRegisters), iRegisterIndex := 151, iBitIndex := 12, xValue := stBunker[3].xVibratorStateRemoteAuto);
FC_ModbusWriteBool(pRegisters := ADR(awModbusInputRegisters), iRegisterIndex := 151, iBitIndex := 13, xValue := stBunker[3].xVibratorStateRemoteManual);
FC_ModbusWriteBool(pRegisters := ADR(awModbusInputRegisters), iRegisterIndex := 151, iBitIndex := 14, xValue := stBunker[3].xVibratorStateRemoteRepair);

FC_ModbusWriteReal(pRegisters := ADR(awModbusInputRegisters), iRegisterIndex := 152, rValue := stBunker[3].rWeight);
FC_ModbusWriteReal(pRegisters := ADR(awModbusInputRegisters), iRegisterIndex := 154, rValue := stBunker[3].rProportionActual);
FC_ModbusWriteReal(pRegisters := ADR(awModbusInputRegisters), iRegisterIndex := 158, rValue := stBunker[3].cmdDumpingPrecent);
FC_ModbusWriteReal(pRegisters := ADR(awModbusInputRegisters), iRegisterIndex := 160, rValue := stBunker[3].MotorVibrator[1].VFD.qrOutFrequency);
FC_ModbusWriteReal(pRegisters := ADR(awModbusInputRegisters), iRegisterIndex := 162, rValue := stBunker[3].MotorVibrator[1].VFD.rActualFrequency);
FC_ModbusWriteReal(pRegisters := ADR(awModbusInputRegisters), iRegisterIndex := 164, rValue := stBunker[3].MotorVibrator[1].VFD.wMotorCurrent.rTag);
FC_ModbusWriteReal(pRegisters := ADR(awModbusInputRegisters), iRegisterIndex := 166, rValue := stBunker[3].MotorVibrator[2].VFD.qrOutFrequency);
FC_ModbusWriteReal(pRegisters := ADR(awModbusInputRegisters), iRegisterIndex := 168, rValue := stBunker[3].MotorVibrator[2].VFD.rActualFrequency);
FC_ModbusWriteReal(pRegisters := ADR(awModbusInputRegisters), iRegisterIndex := 170, rValue := stBunker[3].MotorVibrator[2].VFD.wMotorCurrent.rTag);
FC_ModbusWriteReal(pRegisters := ADR(awModbusInputRegisters), iRegisterIndex := 172, rValue := stBunker[3].MotorVibrator[3].VFD.qrOutFrequency);
FC_ModbusWriteReal(pRegisters := ADR(awModbusInputRegisters), iRegisterIndex := 174, rValue := stBunker[3].MotorVibrator[3].VFD.rActualFrequency);
FC_ModbusWriteReal(pRegisters := ADR(awModbusInputRegisters), iRegisterIndex := 176, rValue := stBunker[3].MotorVibrator[3].VFD.wMotorCurrent.rTag);
FC_ModbusWriteReal(pRegisters := ADR(awModbusInputRegisters), iRegisterIndex := 178, rValue := stBunker[3].MotorVibrator[4].VFD.qrOutFrequency);
FC_ModbusWriteReal(pRegisters := ADR(awModbusInputRegisters), iRegisterIndex := 180, rValue := stBunker[3].MotorVibrator[4].VFD.rActualFrequency);
FC_ModbusWriteReal(pRegisters := ADR(awModbusInputRegisters), iRegisterIndex := 182, rValue := stBunker[3].MotorVibrator[4].VFD.wMotorCurrent.rTag);
FC_ModbusWriteReal(pRegisters := ADR(awModbusInputRegisters), iRegisterIndex := 184, rValue := stBunker[3].MotorVibFeeder[1].VFD.qrOutFrequency);
FC_ModbusWriteReal(pRegisters := ADR(awModbusInputRegisters), iRegisterIndex := 186, rValue := stBunker[3].MotorVibFeeder[1].VFD.rActualFrequency);
FC_ModbusWriteReal(pRegisters := ADR(awModbusInputRegisters), iRegisterIndex := 188, rValue := stBunker[3].MotorVibFeeder[1].VFD.wMotorCurrent.rTag);
FC_ModbusWriteReal(pRegisters := ADR(awModbusInputRegisters), iRegisterIndex := 190, rValue := stBunker[3].MotorVibFeeder[2].VFD.qrOutFrequency);
FC_ModbusWriteReal(pRegisters := ADR(awModbusInputRegisters), iRegisterIndex := 192, rValue := stBunker[3].MotorVibFeeder[2].VFD.rActualFrequency);
FC_ModbusWriteReal(pRegisters := ADR(awModbusInputRegisters), iRegisterIndex := 194, rValue := stBunker[3].MotorVibFeeder[2].VFD.wMotorCurrent.rTag);
FC_ModbusWriteReal(pRegisters := ADR(awModbusInputRegisters), iRegisterIndex := 196, rValue := stBunker[3].MotorVibFeeder[1].rTempBearing[1]);
FC_ModbusWriteReal(pRegisters := ADR(awModbusInputRegisters), iRegisterIndex := 198, rValue := stBunker[3].MotorVibFeeder[1].rTempBearing[2]);
FC_ModbusWriteReal(pRegisters := ADR(awModbusInputRegisters), iRegisterIndex := 200, rValue := stBunker[3].MotorVibFeeder[2].rTempBearing[1]);
FC_ModbusWriteReal(pRegisters := ADR(awModbusInputRegisters), iRegisterIndex := 202, rValue := stBunker[3].MotorVibFeeder[2].rTempBearing[2]);

FC_ModbusWriteUInt(pRegisters := ADR(awModbusInputRegisters), iRegisterIndex := 204, uValue := eBunkerStageToSCADA[3]);

// Отвалообразователь - Конвейер (210-239)
// Регистры 210-211: BOOL флаги статусов отвалообразователя
FC_ModbusWriteBool(pRegisters := ADR(awModbusInputRegisters), iRegisterIndex := 210, iBitIndex := 0, xValue := stDumper.xStateWarning);
FC_ModbusWriteBool(pRegisters := ADR(awModbusInputRegisters), iRegisterIndex := 210, iBitIndex := 1, xValue := stDumper.xStateFailure);
FC_ModbusWriteBool(pRegisters := ADR(awModbusInputRegisters), iRegisterIndex := 210, iBitIndex := 2, xValue := stDumper.xStateEnable);
FC_ModbusWriteBool(pRegisters := ADR(awModbusInputRegisters), iRegisterIndex := 210, iBitIndex := 3, xValue := stDumper.xStateStarting);
FC_ModbusWriteBool(pRegisters := ADR(awModbusInputRegisters), iRegisterIndex := 210, iBitIndex := 7, xValue := stDumper.fbBtnRemoteMode.qxSignal);
FC_ModbusWriteBool(pRegisters := ADR(awModbusInputRegisters), iRegisterIndex := 210, iBitIndex := 9, xValue := stDumper.xSoundAlarm);

// Регистр 211: дополнительные сигналы обратной связи отвалообразователя
FC_ModbusWriteBool(pRegisters := ADR(awModbusInputRegisters), iRegisterIndex := 211, iBitIndex := 12, xValue := stDumper.xStateRemoteAuto);
FC_ModbusWriteBool(pRegisters := ADR(awModbusInputRegisters), iRegisterIndex := 211, iBitIndex := 13, xValue := stDumper.xStateRemoteManual);
FC_ModbusWriteBool(pRegisters := ADR(awModbusInputRegisters), iRegisterIndex := 211, iBitIndex := 14, xValue := stDumper.xStateRemoteRepair);

FC_ModbusWriteReal(pRegisters := ADR(awModbusInputRegisters), iRegisterIndex := 212, rValue := stDumper.MotorConveyor[1].VFD.qrOutFrequency);
FC_ModbusWriteReal(pRegisters := ADR(awModbusInputRegisters), iRegisterIndex := 214, rValue := stDumper.MotorConveyor[1].VFD.rActualFrequency);
FC_ModbusWriteReal(pRegisters := ADR(awModbusInputRegisters), iRegisterIndex := 216, rValue := stDumper.MotorConveyor[1].VFD.wMotorCurrent.rTag);
FC_ModbusWriteReal(pRegisters := ADR(awModbusInputRegisters), iRegisterIndex := 218, rValue := stDumper.MotorConveyor[2].VFD.qrOutFrequency);
FC_ModbusWriteReal(pRegisters := ADR(awModbusInputRegisters), iRegisterIndex := 220, rValue := stDumper.MotorConveyor[2].VFD.rActualFrequency);
FC_ModbusWriteReal(pRegisters := ADR(awModbusInputRegisters), iRegisterIndex := 222, rValue := stDumper.MotorConveyor[2].VFD.wMotorCurrent.rTag);

FC_ModbusWriteUInt(pRegisters := ADR(awModbusInputRegisters), iRegisterIndex := 230, uValue := eDumperStageToSCADA);

// Отвалообразователь - Поворот (240-269)
// Регистры 240-241: BOOL флаги управления поворотом (данные перенесены в DI модули)

FC_ModbusWriteReal(pRegisters := ADR(awModbusInputRegisters), iRegisterIndex := 242, rValue := stDumper.MotorRotation[1].VFD.qrOutFrequency);
FC_ModbusWriteReal(pRegisters := ADR(awModbusInputRegisters), iRegisterIndex := 244, rValue := stDumper.MotorRotation[1].VFD.rActualFrequency);
FC_ModbusWriteReal(pRegisters := ADR(awModbusInputRegisters), iRegisterIndex := 246, rValue := stDumper.MotorRotation[1].VFD.wMotorCurrent.rTag);
FC_ModbusWriteReal(pRegisters := ADR(awModbusInputRegisters), iRegisterIndex := 248, rValue := stDumper.MotorRotation[2].VFD.qrOutFrequency);
FC_ModbusWriteReal(pRegisters := ADR(awModbusInputRegisters), iRegisterIndex := 250, rValue := stDumper.MotorRotation[2].VFD.rActualFrequency);
FC_ModbusWriteReal(pRegisters := ADR(awModbusInputRegisters), iRegisterIndex := 252, rValue := stDumper.MotorRotation[2].VFD.wMotorCurrent.rTag);

// Конвейер (270-299)
// Регистры 270-271: BOOL флаги статусов конвейера
FC_ModbusWriteBool(pRegisters := ADR(awModbusInputRegisters), iRegisterIndex := 270, iBitIndex := 0, xValue := stConveyor.xStateWarning);
FC_ModbusWriteBool(pRegisters := ADR(awModbusInputRegisters), iRegisterIndex := 270, iBitIndex := 1, xValue := stConveyor.xStateFailure);
FC_ModbusWriteBool(pRegisters := ADR(awModbusInputRegisters), iRegisterIndex := 270, iBitIndex := 2, xValue := stConveyor.xStateEnable);
FC_ModbusWriteBool(pRegisters := ADR(awModbusInputRegisters), iRegisterIndex := 270, iBitIndex := 3, xValue := stConveyor.xStateStarting);
FC_ModbusWriteBool(pRegisters := ADR(awModbusInputRegisters), iRegisterIndex := 270, iBitIndex := 8, xValue := stConveyor.xSoundAlarm);

// Регистр 271: дополнительные сигналы обратной связи конвейера
FC_ModbusWriteBool(pRegisters := ADR(awModbusInputRegisters), iRegisterIndex := 271, iBitIndex := 12, xValue := stConveyor.xStateRemoteAuto);
FC_ModbusWriteBool(pRegisters := ADR(awModbusInputRegisters), iRegisterIndex := 271, iBitIndex := 13, xValue := stConveyor.xStateRemoteManual);
FC_ModbusWriteBool(pRegisters := ADR(awModbusInputRegisters), iRegisterIndex := 271, iBitIndex := 14, xValue := stConveyor.xStateRemoteRepair);

FC_ModbusWriteReal(pRegisters := ADR(awModbusInputRegisters), iRegisterIndex := 272, rValue := stConveyor.MotorConveyor[1].VFD.qrOutFrequency);
FC_ModbusWriteReal(pRegisters := ADR(awModbusInputRegisters), iRegisterIndex := 274, rValue := stConveyor.MotorConveyor[1].VFD.rActualFrequency);
FC_ModbusWriteReal(pRegisters := ADR(awModbusInputRegisters), iRegisterIndex := 276, rValue := stConveyor.MotorConveyor[1].VFD.wMotorCurrent.rTag);
FC_ModbusWriteReal(pRegisters := ADR(awModbusInputRegisters), iRegisterIndex := 278, rValue := stConveyor.MotorConveyor[2].VFD.qrOutFrequency);
FC_ModbusWriteReal(pRegisters := ADR(awModbusInputRegisters), iRegisterIndex := 280, rValue := stConveyor.MotorConveyor[2].VFD.rActualFrequency);
FC_ModbusWriteReal(pRegisters := ADR(awModbusInputRegisters), iRegisterIndex := 282, rValue := stConveyor.MotorConveyor[2].VFD.wMotorCurrent.rTag);

// Регистры 284-289: Конвейерные весы (накопительные веса под бункерами)
FC_ModbusWriteReal(pRegisters := ADR(awModbusInputRegisters), iRegisterIndex := 284, rValue := stBunker[1].rWeightUnderBunker);
FC_ModbusWriteReal(pRegisters := ADR(awModbusInputRegisters), iRegisterIndex := 286, rValue := stBunker[2].rWeightUnderBunker);
FC_ModbusWriteReal(pRegisters := ADR(awModbusInputRegisters), iRegisterIndex := 288, rValue := stBunker[3].rWeightUnderBunker);

FC_ModbusWriteUInt(pRegisters := ADR(awModbusInputRegisters), iRegisterIndex := 290, uValue := eConveyorStageToSCADA);

// DI MODULES MAPPING (300-399)

// Модуль DI1 (300-301): Бункер 1 - Вибропитатели и вибраторы
FC_ModbusWriteBool(pRegisters := ADR(awModbusInputRegisters), iRegisterIndex := 300, iBitIndex := 0, xValue := stBunker[1].fbStateHatch.qxSignal);
FC_ModbusWriteBool(pRegisters := ADR(awModbusInputRegisters), iRegisterIndex := 300, iBitIndex := 1, xValue := stBunker[1].MotorVibFeeder[1].VFD.fbStateRdyToStart.qxSignal);
FC_ModbusWriteBool(pRegisters := ADR(awModbusInputRegisters), iRegisterIndex := 300, iBitIndex := 2, xValue := stBunker[1].MotorVibFeeder[1].VFD.fbStateIsWorking.qxSignal);
FC_ModbusWriteBool(pRegisters := ADR(awModbusInputRegisters), iRegisterIndex := 300, iBitIndex := 3, xValue := stBunker[1].MotorVibFeeder[1].VFD.fbStateFailure.qxSignal);
FC_ModbusWriteBool(pRegisters := ADR(awModbusInputRegisters), iRegisterIndex := 300, iBitIndex := 4, xValue := stBunker[1].MotorVibFeeder[1].fbStateQF.qxSignal);
FC_ModbusWriteBool(pRegisters := ADR(awModbusInputRegisters), iRegisterIndex := 300, iBitIndex := 5, xValue := stBunker[1].MotorVibFeeder[1].fbStateKM.qxSignal);
FC_ModbusWriteBool(pRegisters := ADR(awModbusInputRegisters), iRegisterIndex := 300, iBitIndex := 6, xValue := stBunker[1].MotorVibFeeder[2].VFD.fbStateRdyToStart.qxSignal);
FC_ModbusWriteBool(pRegisters := ADR(awModbusInputRegisters), iRegisterIndex := 300, iBitIndex := 7, xValue := stBunker[1].MotorVibFeeder[2].VFD.fbStateIsWorking.qxSignal);
FC_ModbusWriteBool(pRegisters := ADR(awModbusInputRegisters), iRegisterIndex := 300, iBitIndex := 8, xValue := stBunker[1].MotorVibFeeder[2].VFD.fbStateFailure.qxSignal);
FC_ModbusWriteBool(pRegisters := ADR(awModbusInputRegisters), iRegisterIndex := 300, iBitIndex := 9, xValue := stBunker[1].MotorVibFeeder[2].fbStateQF.qxSignal);
FC_ModbusWriteBool(pRegisters := ADR(awModbusInputRegisters), iRegisterIndex := 300, iBitIndex := 10, xValue := stBunker[1].MotorVibFeeder[2].fbStateKM.qxSignal);
FC_ModbusWriteBool(pRegisters := ADR(awModbusInputRegisters), iRegisterIndex := 300, iBitIndex := 11, xValue := stBunker[1].MotorVibrator[1].VFD.fbStateRdyToStart.qxSignal);
FC_ModbusWriteBool(pRegisters := ADR(awModbusInputRegisters), iRegisterIndex := 300, iBitIndex := 12, xValue := stBunker[1].MotorVibrator[1].VFD.fbStateIsWorking.qxSignal);
FC_ModbusWriteBool(pRegisters := ADR(awModbusInputRegisters), iRegisterIndex := 300, iBitIndex := 13, xValue := stBunker[1].MotorVibrator[1].VFD.fbStateFailure.qxSignal);
FC_ModbusWriteBool(pRegisters := ADR(awModbusInputRegisters), iRegisterIndex := 300, iBitIndex := 14, xValue := stBunker[1].MotorVibrator[1].fbStateQF.qxSignal);
FC_ModbusWriteBool(pRegisters := ADR(awModbusInputRegisters), iRegisterIndex := 300, iBitIndex := 15, xValue := stBunker[1].MotorVibrator[1].fbStateKM.qxSignal);

FC_ModbusWriteBool(pRegisters := ADR(awModbusInputRegisters), iRegisterIndex := 301, iBitIndex := 0, xValue := stBunker[1].MotorVibrator[2].VFD.fbStateRdyToStart.qxSignal);
FC_ModbusWriteBool(pRegisters := ADR(awModbusInputRegisters), iRegisterIndex := 301, iBitIndex := 1, xValue := stBunker[1].MotorVibrator[2].VFD.fbStateIsWorking.qxSignal);
FC_ModbusWriteBool(pRegisters := ADR(awModbusInputRegisters), iRegisterIndex := 301, iBitIndex := 2, xValue := stBunker[1].MotorVibrator[2].VFD.fbStateFailure.qxSignal);
FC_ModbusWriteBool(pRegisters := ADR(awModbusInputRegisters), iRegisterIndex := 301, iBitIndex := 3, xValue := stBunker[1].MotorVibrator[2].fbStateQF.qxSignal);
FC_ModbusWriteBool(pRegisters := ADR(awModbusInputRegisters), iRegisterIndex := 301, iBitIndex := 4, xValue := stBunker[1].MotorVibrator[2].fbStateKM.qxSignal);
FC_ModbusWriteBool(pRegisters := ADR(awModbusInputRegisters), iRegisterIndex := 301, iBitIndex := 5, xValue := stBunker[1].MotorVibrator[3].VFD.fbStateRdyToStart.qxSignal);
FC_ModbusWriteBool(pRegisters := ADR(awModbusInputRegisters), iRegisterIndex := 301, iBitIndex := 6, xValue := stBunker[1].MotorVibrator[3].VFD.fbStateIsWorking.qxSignal);
FC_ModbusWriteBool(pRegisters := ADR(awModbusInputRegisters), iRegisterIndex := 301, iBitIndex := 7, xValue := stBunker[1].MotorVibrator[3].VFD.fbStateFailure.qxSignal);
FC_ModbusWriteBool(pRegisters := ADR(awModbusInputRegisters), iRegisterIndex := 301, iBitIndex := 8, xValue := stBunker[1].MotorVibrator[3].fbStateQF.qxSignal);
FC_ModbusWriteBool(pRegisters := ADR(awModbusInputRegisters), iRegisterIndex := 301, iBitIndex := 9, xValue := stBunker[1].MotorVibrator[3].fbStateKM.qxSignal);
FC_ModbusWriteBool(pRegisters := ADR(awModbusInputRegisters), iRegisterIndex := 301, iBitIndex := 10, xValue := stBunker[1].MotorVibrator[4].VFD.fbStateRdyToStart.qxSignal);
FC_ModbusWriteBool(pRegisters := ADR(awModbusInputRegisters), iRegisterIndex := 301, iBitIndex := 11, xValue := stBunker[1].MotorVibrator[4].VFD.fbStateIsWorking.qxSignal);
FC_ModbusWriteBool(pRegisters := ADR(awModbusInputRegisters), iRegisterIndex := 301, iBitIndex := 12, xValue := stBunker[1].MotorVibrator[4].VFD.fbStateFailure.qxSignal);
FC_ModbusWriteBool(pRegisters := ADR(awModbusInputRegisters), iRegisterIndex := 301, iBitIndex := 13, xValue := stBunker[1].MotorVibrator[4].fbStateQF.qxSignal);
FC_ModbusWriteBool(pRegisters := ADR(awModbusInputRegisters), iRegisterIndex := 301, iBitIndex := 14, xValue := stBunker[1].MotorVibrator[4].fbStateKM.qxSignal);

// Модуль DI2 (302-303): Бункер 2 - Вибропитатели и вибраторы
FC_ModbusWriteBool(pRegisters := ADR(awModbusInputRegisters), iRegisterIndex := 302, iBitIndex := 0, xValue := stBunker[2].fbStateHatch.qxSignal);
FC_ModbusWriteBool(pRegisters := ADR(awModbusInputRegisters), iRegisterIndex := 302, iBitIndex := 1, xValue := stBunker[2].MotorVibFeeder[1].VFD.fbStateRdyToStart.qxSignal);
FC_ModbusWriteBool(pRegisters := ADR(awModbusInputRegisters), iRegisterIndex := 302, iBitIndex := 2, xValue := stBunker[2].MotorVibFeeder[1].VFD.fbStateIsWorking.qxSignal);
FC_ModbusWriteBool(pRegisters := ADR(awModbusInputRegisters), iRegisterIndex := 302, iBitIndex := 3, xValue := stBunker[2].MotorVibFeeder[1].VFD.fbStateFailure.qxSignal);
FC_ModbusWriteBool(pRegisters := ADR(awModbusInputRegisters), iRegisterIndex := 302, iBitIndex := 4, xValue := stBunker[2].MotorVibFeeder[1].fbStateQF.qxSignal);
FC_ModbusWriteBool(pRegisters := ADR(awModbusInputRegisters), iRegisterIndex := 302, iBitIndex := 5, xValue := stBunker[2].MotorVibFeeder[1].fbStateKM.qxSignal);
FC_ModbusWriteBool(pRegisters := ADR(awModbusInputRegisters), iRegisterIndex := 302, iBitIndex := 6, xValue := stBunker[2].MotorVibFeeder[2].VFD.fbStateRdyToStart.qxSignal);
FC_ModbusWriteBool(pRegisters := ADR(awModbusInputRegisters), iRegisterIndex := 302, iBitIndex := 7, xValue := stBunker[2].MotorVibFeeder[2].VFD.fbStateIsWorking.qxSignal);
FC_ModbusWriteBool(pRegisters := ADR(awModbusInputRegisters), iRegisterIndex := 302, iBitIndex := 8, xValue := stBunker[2].MotorVibFeeder[2].VFD.fbStateFailure.qxSignal);
FC_ModbusWriteBool(pRegisters := ADR(awModbusInputRegisters), iRegisterIndex := 302, iBitIndex := 9, xValue := stBunker[2].MotorVibFeeder[2].fbStateQF.qxSignal);
FC_ModbusWriteBool(pRegisters := ADR(awModbusInputRegisters), iRegisterIndex := 302, iBitIndex := 10, xValue := stBunker[2].MotorVibFeeder[2].fbStateKM.qxSignal);
FC_ModbusWriteBool(pRegisters := ADR(awModbusInputRegisters), iRegisterIndex := 302, iBitIndex := 11, xValue := stBunker[2].MotorVibrator[1].VFD.fbStateRdyToStart.qxSignal);
FC_ModbusWriteBool(pRegisters := ADR(awModbusInputRegisters), iRegisterIndex := 302, iBitIndex := 12, xValue := stBunker[2].MotorVibrator[1].VFD.fbStateIsWorking.qxSignal);
FC_ModbusWriteBool(pRegisters := ADR(awModbusInputRegisters), iRegisterIndex := 302, iBitIndex := 13, xValue := stBunker[2].MotorVibrator[1].VFD.fbStateFailure.qxSignal);
FC_ModbusWriteBool(pRegisters := ADR(awModbusInputRegisters), iRegisterIndex := 302, iBitIndex := 14, xValue := stBunker[2].MotorVibrator[1].fbStateQF.qxSignal);
FC_ModbusWriteBool(pRegisters := ADR(awModbusInputRegisters), iRegisterIndex := 302, iBitIndex := 15, xValue := stBunker[2].MotorVibrator[1].fbStateKM.qxSignal);

FC_ModbusWriteBool(pRegisters := ADR(awModbusInputRegisters), iRegisterIndex := 303, iBitIndex := 0, xValue := stBunker[2].MotorVibrator[2].VFD.fbStateRdyToStart.qxSignal);
FC_ModbusWriteBool(pRegisters := ADR(awModbusInputRegisters), iRegisterIndex := 303, iBitIndex := 1, xValue := stBunker[2].MotorVibrator[2].VFD.fbStateIsWorking.qxSignal);
FC_ModbusWriteBool(pRegisters := ADR(awModbusInputRegisters), iRegisterIndex := 303, iBitIndex := 2, xValue := stBunker[2].MotorVibrator[2].VFD.fbStateFailure.qxSignal);
FC_ModbusWriteBool(pRegisters := ADR(awModbusInputRegisters), iRegisterIndex := 303, iBitIndex := 3, xValue := stBunker[2].MotorVibrator[2].fbStateQF.qxSignal);
FC_ModbusWriteBool(pRegisters := ADR(awModbusInputRegisters), iRegisterIndex := 303, iBitIndex := 4, xValue := stBunker[2].MotorVibrator[2].fbStateKM.qxSignal);
FC_ModbusWriteBool(pRegisters := ADR(awModbusInputRegisters), iRegisterIndex := 303, iBitIndex := 5, xValue := stBunker[2].MotorVibrator[3].VFD.fbStateRdyToStart.qxSignal);
FC_ModbusWriteBool(pRegisters := ADR(awModbusInputRegisters), iRegisterIndex := 303, iBitIndex := 6, xValue := stBunker[2].MotorVibrator[3].VFD.fbStateIsWorking.qxSignal);
FC_ModbusWriteBool(pRegisters := ADR(awModbusInputRegisters), iRegisterIndex := 303, iBitIndex := 7, xValue := stBunker[2].MotorVibrator[3].VFD.fbStateFailure.qxSignal);
FC_ModbusWriteBool(pRegisters := ADR(awModbusInputRegisters), iRegisterIndex := 303, iBitIndex := 8, xValue := stBunker[2].MotorVibrator[3].fbStateQF.qxSignal);
FC_ModbusWriteBool(pRegisters := ADR(awModbusInputRegisters), iRegisterIndex := 303, iBitIndex := 9, xValue := stBunker[2].MotorVibrator[3].fbStateKM.qxSignal);
FC_ModbusWriteBool(pRegisters := ADR(awModbusInputRegisters), iRegisterIndex := 303, iBitIndex := 10, xValue := stBunker[2].MotorVibrator[4].VFD.fbStateRdyToStart.qxSignal);
FC_ModbusWriteBool(pRegisters := ADR(awModbusInputRegisters), iRegisterIndex := 303, iBitIndex := 11, xValue := stBunker[2].MotorVibrator[4].VFD.fbStateIsWorking.qxSignal);
FC_ModbusWriteBool(pRegisters := ADR(awModbusInputRegisters), iRegisterIndex := 303, iBitIndex := 12, xValue := stBunker[2].MotorVibrator[4].VFD.fbStateFailure.qxSignal);
FC_ModbusWriteBool(pRegisters := ADR(awModbusInputRegisters), iRegisterIndex := 303, iBitIndex := 13, xValue := stBunker[2].MotorVibrator[4].fbStateQF.qxSignal);
FC_ModbusWriteBool(pRegisters := ADR(awModbusInputRegisters), iRegisterIndex := 303, iBitIndex := 14, xValue := stBunker[2].MotorVibrator[4].fbStateKM.qxSignal);

// Модуль DI3 (304-305): Бункер 3 - Вибропитатели и вибраторы
FC_ModbusWriteBool(pRegisters := ADR(awModbusInputRegisters), iRegisterIndex := 304, iBitIndex := 0, xValue := stBunker[3].fbStateHatch.qxSignal);
FC_ModbusWriteBool(pRegisters := ADR(awModbusInputRegisters), iRegisterIndex := 304, iBitIndex := 1, xValue := stBunker[3].MotorVibFeeder[1].VFD.fbStateRdyToStart.qxSignal);
FC_ModbusWriteBool(pRegisters := ADR(awModbusInputRegisters), iRegisterIndex := 304, iBitIndex := 2, xValue := stBunker[3].MotorVibFeeder[1].VFD.fbStateIsWorking.qxSignal);
FC_ModbusWriteBool(pRegisters := ADR(awModbusInputRegisters), iRegisterIndex := 304, iBitIndex := 3, xValue := stBunker[3].MotorVibFeeder[1].VFD.fbStateFailure.qxSignal);
FC_ModbusWriteBool(pRegisters := ADR(awModbusInputRegisters), iRegisterIndex := 304, iBitIndex := 4, xValue := stBunker[3].MotorVibFeeder[1].fbStateQF.qxSignal);
FC_ModbusWriteBool(pRegisters := ADR(awModbusInputRegisters), iRegisterIndex := 304, iBitIndex := 5, xValue := stBunker[3].MotorVibFeeder[1].fbStateKM.qxSignal);
FC_ModbusWriteBool(pRegisters := ADR(awModbusInputRegisters), iRegisterIndex := 304, iBitIndex := 6, xValue := stBunker[3].MotorVibFeeder[2].VFD.fbStateRdyToStart.qxSignal);
FC_ModbusWriteBool(pRegisters := ADR(awModbusInputRegisters), iRegisterIndex := 304, iBitIndex := 7, xValue := stBunker[3].MotorVibFeeder[2].VFD.fbStateIsWorking.qxSignal);
FC_ModbusWriteBool(pRegisters := ADR(awModbusInputRegisters), iRegisterIndex := 304, iBitIndex := 8, xValue := stBunker[3].MotorVibFeeder[2].VFD.fbStateFailure.qxSignal);
FC_ModbusWriteBool(pRegisters := ADR(awModbusInputRegisters), iRegisterIndex := 304, iBitIndex := 9, xValue := stBunker[3].MotorVibFeeder[2].fbStateQF.qxSignal);
FC_ModbusWriteBool(pRegisters := ADR(awModbusInputRegisters), iRegisterIndex := 304, iBitIndex := 10, xValue := stBunker[3].MotorVibFeeder[2].fbStateKM.qxSignal);
FC_ModbusWriteBool(pRegisters := ADR(awModbusInputRegisters), iRegisterIndex := 304, iBitIndex := 11, xValue := stBunker[3].MotorVibrator[1].VFD.fbStateRdyToStart.qxSignal);
FC_ModbusWriteBool(pRegisters := ADR(awModbusInputRegisters), iRegisterIndex := 304, iBitIndex := 12, xValue := stBunker[3].MotorVibrator[1].VFD.fbStateIsWorking.qxSignal);
FC_ModbusWriteBool(pRegisters := ADR(awModbusInputRegisters), iRegisterIndex := 304, iBitIndex := 13, xValue := stBunker[3].MotorVibrator[1].VFD.fbStateFailure.qxSignal);
FC_ModbusWriteBool(pRegisters := ADR(awModbusInputRegisters), iRegisterIndex := 304, iBitIndex := 14, xValue := stBunker[3].MotorVibrator[1].fbStateQF.qxSignal);
FC_ModbusWriteBool(pRegisters := ADR(awModbusInputRegisters), iRegisterIndex := 304, iBitIndex := 15, xValue := stBunker[3].MotorVibrator[1].fbStateKM.qxSignal);

FC_ModbusWriteBool(pRegisters := ADR(awModbusInputRegisters), iRegisterIndex := 305, iBitIndex := 0, xValue := stBunker[3].MotorVibrator[2].VFD.fbStateRdyToStart.qxSignal);
FC_ModbusWriteBool(pRegisters := ADR(awModbusInputRegisters), iRegisterIndex := 305, iBitIndex := 1, xValue := stBunker[3].MotorVibrator[2].VFD.fbStateIsWorking.qxSignal);
FC_ModbusWriteBool(pRegisters := ADR(awModbusInputRegisters), iRegisterIndex := 305, iBitIndex := 2, xValue := stBunker[3].MotorVibrator[2].VFD.fbStateFailure.qxSignal);
FC_ModbusWriteBool(pRegisters := ADR(awModbusInputRegisters), iRegisterIndex := 305, iBitIndex := 3, xValue := stBunker[3].MotorVibrator[2].fbStateQF.qxSignal);
FC_ModbusWriteBool(pRegisters := ADR(awModbusInputRegisters), iRegisterIndex := 305, iBitIndex := 4, xValue := stBunker[3].MotorVibrator[2].fbStateKM.qxSignal);
FC_ModbusWriteBool(pRegisters := ADR(awModbusInputRegisters), iRegisterIndex := 305, iBitIndex := 5, xValue := stBunker[3].MotorVibrator[3].VFD.fbStateRdyToStart.qxSignal);
FC_ModbusWriteBool(pRegisters := ADR(awModbusInputRegisters), iRegisterIndex := 305, iBitIndex := 6, xValue := stBunker[3].MotorVibrator[3].VFD.fbStateIsWorking.qxSignal);
FC_ModbusWriteBool(pRegisters := ADR(awModbusInputRegisters), iRegisterIndex := 305, iBitIndex := 7, xValue := stBunker[3].MotorVibrator[3].VFD.fbStateFailure.qxSignal);
FC_ModbusWriteBool(pRegisters := ADR(awModbusInputRegisters), iRegisterIndex := 305, iBitIndex := 8, xValue := stBunker[3].MotorVibrator[3].fbStateQF.qxSignal);
FC_ModbusWriteBool(pRegisters := ADR(awModbusInputRegisters), iRegisterIndex := 305, iBitIndex := 9, xValue := stBunker[3].MotorVibrator[3].fbStateKM.qxSignal);
FC_ModbusWriteBool(pRegisters := ADR(awModbusInputRegisters), iRegisterIndex := 305, iBitIndex := 10, xValue := stBunker[3].MotorVibrator[4].VFD.fbStateRdyToStart.qxSignal);
FC_ModbusWriteBool(pRegisters := ADR(awModbusInputRegisters), iRegisterIndex := 305, iBitIndex := 11, xValue := stBunker[3].MotorVibrator[4].VFD.fbStateIsWorking.qxSignal);
FC_ModbusWriteBool(pRegisters := ADR(awModbusInputRegisters), iRegisterIndex := 305, iBitIndex := 12, xValue := stBunker[3].MotorVibrator[4].VFD.fbStateFailure.qxSignal);
FC_ModbusWriteBool(pRegisters := ADR(awModbusInputRegisters), iRegisterIndex := 305, iBitIndex := 13, xValue := stBunker[3].MotorVibrator[4].fbStateQF.qxSignal);
FC_ModbusWriteBool(pRegisters := ADR(awModbusInputRegisters), iRegisterIndex := 305, iBitIndex := 14, xValue := stBunker[3].MotorVibrator[4].fbStateKM.qxSignal);

// Модуль DI4 (306-307): Конвейер - Датчики и моторы
FC_ModbusWriteBool(pRegisters := ADR(awModbusInputRegisters), iRegisterIndex := 306, iBitIndex := 0, xValue := stConveyor.fbSQ_IsOk[1].qxSignal);
FC_ModbusWriteBool(pRegisters := ADR(awModbusInputRegisters), iRegisterIndex := 306, iBitIndex := 1, xValue := stConveyor.fbSQ_IsOk[2].qxSignal);
FC_ModbusWriteBool(pRegisters := ADR(awModbusInputRegisters), iRegisterIndex := 306, iBitIndex := 2, xValue := stConveyor.fbHQ_IsOk[1].qxSignal);
FC_ModbusWriteBool(pRegisters := ADR(awModbusInputRegisters), iRegisterIndex := 306, iBitIndex := 3, xValue := stConveyor.fbHQ_IsOk[2].qxSignal);
FC_ModbusWriteBool(pRegisters := ADR(awModbusInputRegisters), iRegisterIndex := 306, iBitIndex := 4, xValue := stConveyor.fbHQ_IsOk[3].qxSignal);
FC_ModbusWriteBool(pRegisters := ADR(awModbusInputRegisters), iRegisterIndex := 306, iBitIndex := 5, xValue := stConveyor.fbHQ_IsOk[4].qxSignal);
FC_ModbusWriteBool(pRegisters := ADR(awModbusInputRegisters), iRegisterIndex := 306, iBitIndex := 6, xValue := stConveyor.fbZQWarning[1].qxSignal);
FC_ModbusWriteBool(pRegisters := ADR(awModbusInputRegisters), iRegisterIndex := 306, iBitIndex := 7, xValue := stConveyor.fbZQAlarm[1].qxSignal);
FC_ModbusWriteBool(pRegisters := ADR(awModbusInputRegisters), iRegisterIndex := 306, iBitIndex := 8, xValue := stConveyor.fbZQWarning[2].qxSignal);
FC_ModbusWriteBool(pRegisters := ADR(awModbusInputRegisters), iRegisterIndex := 306, iBitIndex := 9, xValue := stConveyor.fbZQAlarm[2].qxSignal);
FC_ModbusWriteBool(pRegisters := ADR(awModbusInputRegisters), iRegisterIndex := 306, iBitIndex := 10, xValue := stConveyor.fbZQWarning[3].qxSignal);
FC_ModbusWriteBool(pRegisters := ADR(awModbusInputRegisters), iRegisterIndex := 306, iBitIndex := 11, xValue := stConveyor.fbZQAlarm[3].qxSignal);
FC_ModbusWriteBool(pRegisters := ADR(awModbusInputRegisters), iRegisterIndex := 306, iBitIndex := 12, xValue := stConveyor.fbZQWarning[4].qxSignal);
FC_ModbusWriteBool(pRegisters := ADR(awModbusInputRegisters), iRegisterIndex := 306, iBitIndex := 13, xValue := stConveyor.fbZQAlarm[4].qxSignal);
FC_ModbusWriteBool(pRegisters := ADR(awModbusInputRegisters), iRegisterIndex := 306, iBitIndex := 14, xValue := stConveyor.fbGS1.qxSignal);
FC_ModbusWriteBool(pRegisters := ADR(awModbusInputRegisters), iRegisterIndex := 306, iBitIndex := 15, xValue := stConveyor.fbYS1.qxSignal);

FC_ModbusWriteBool(pRegisters := ADR(awModbusInputRegisters), iRegisterIndex := 307, iBitIndex := 0, xValue := stConveyor.fbQR[1].qxSignal);
FC_ModbusWriteBool(pRegisters := ADR(awModbusInputRegisters), iRegisterIndex := 307, iBitIndex := 1, xValue := stConveyor.fbQR[2].qxSignal);
FC_ModbusWriteBool(pRegisters := ADR(awModbusInputRegisters), iRegisterIndex := 307, iBitIndex := 2, xValue := stConveyor.fbYE1.qxSignal);
FC_ModbusWriteBool(pRegisters := ADR(awModbusInputRegisters), iRegisterIndex := 307, iBitIndex := 3, xValue := stConveyor.MotorConveyor[1].fbStatorOverheat.qxSignal);
FC_ModbusWriteBool(pRegisters := ADR(awModbusInputRegisters), iRegisterIndex := 307, iBitIndex := 4, xValue := stConveyor.MotorConveyor[2].fbStatorOverheat.qxSignal);
FC_ModbusWriteBool(pRegisters := ADR(awModbusInputRegisters), iRegisterIndex := 307, iBitIndex := 5, xValue := stConveyor.MotorConveyor[1].VFD.fbStateRdyToStart.qxSignal);
FC_ModbusWriteBool(pRegisters := ADR(awModbusInputRegisters), iRegisterIndex := 307, iBitIndex := 6, xValue := stConveyor.MotorConveyor[1].VFD.fbStateIsWorking.qxSignal);
FC_ModbusWriteBool(pRegisters := ADR(awModbusInputRegisters), iRegisterIndex := 307, iBitIndex := 7, xValue := stConveyor.MotorConveyor[1].VFD.fbStateFailure.qxSignal);
FC_ModbusWriteBool(pRegisters := ADR(awModbusInputRegisters), iRegisterIndex := 307, iBitIndex := 8, xValue := stConveyor.MotorConveyor[1].fbStateQF.qxSignal);
FC_ModbusWriteBool(pRegisters := ADR(awModbusInputRegisters), iRegisterIndex := 307, iBitIndex := 9, xValue := stConveyor.MotorConveyor[1].fbStateKM.qxSignal);
FC_ModbusWriteBool(pRegisters := ADR(awModbusInputRegisters), iRegisterIndex := 307, iBitIndex := 10, xValue := stConveyor.MotorConveyor[2].VFD.fbStateRdyToStart.qxSignal);
FC_ModbusWriteBool(pRegisters := ADR(awModbusInputRegisters), iRegisterIndex := 307, iBitIndex := 11, xValue := stConveyor.MotorConveyor[2].VFD.fbStateIsWorking.qxSignal);
FC_ModbusWriteBool(pRegisters := ADR(awModbusInputRegisters), iRegisterIndex := 307, iBitIndex := 12, xValue := stConveyor.MotorConveyor[2].VFD.fbStateFailure.qxSignal);
FC_ModbusWriteBool(pRegisters := ADR(awModbusInputRegisters), iRegisterIndex := 307, iBitIndex := 13, xValue := stConveyor.MotorConveyor[2].fbStateQF.qxSignal);
FC_ModbusWriteBool(pRegisters := ADR(awModbusInputRegisters), iRegisterIndex := 307, iBitIndex := 14, xValue := stConveyor.MotorConveyor[2].fbStateKM.qxSignal);

// Модуль DI5 (308-309): Отвалообразователь - Датчики и перегрев
FC_ModbusWriteBool(pRegisters := ADR(awModbusInputRegisters), iRegisterIndex := 308, iBitIndex := 0, xValue := stDumper.fbSQ_IsOk[1].qxSignal);
FC_ModbusWriteBool(pRegisters := ADR(awModbusInputRegisters), iRegisterIndex := 308, iBitIndex := 1, xValue := stDumper.fbSQ_IsOk[2].qxSignal);
FC_ModbusWriteBool(pRegisters := ADR(awModbusInputRegisters), iRegisterIndex := 308, iBitIndex := 2, xValue := stDumper.fbHQ_IsOk[1].qxSignal);
FC_ModbusWriteBool(pRegisters := ADR(awModbusInputRegisters), iRegisterIndex := 308, iBitIndex := 3, xValue := stDumper.fbHQ_IsOk[2].qxSignal);
FC_ModbusWriteBool(pRegisters := ADR(awModbusInputRegisters), iRegisterIndex := 308, iBitIndex := 4, xValue := stDumper.fbHQ_IsOk[3].qxSignal);
FC_ModbusWriteBool(pRegisters := ADR(awModbusInputRegisters), iRegisterIndex := 308, iBitIndex := 5, xValue := stDumper.fbHQ_IsOk[4].qxSignal);
FC_ModbusWriteBool(pRegisters := ADR(awModbusInputRegisters), iRegisterIndex := 308, iBitIndex := 6, xValue := stDumper.fbZQWarning[1].qxSignal);
FC_ModbusWriteBool(pRegisters := ADR(awModbusInputRegisters), iRegisterIndex := 308, iBitIndex := 7, xValue := stDumper.fbZQAlarm[1].qxSignal);
FC_ModbusWriteBool(pRegisters := ADR(awModbusInputRegisters), iRegisterIndex := 308, iBitIndex := 8, xValue := stDumper.fbZQWarning[2].qxSignal);
FC_ModbusWriteBool(pRegisters := ADR(awModbusInputRegisters), iRegisterIndex := 308, iBitIndex := 9, xValue := stDumper.fbZQAlarm[2].qxSignal);
FC_ModbusWriteBool(pRegisters := ADR(awModbusInputRegisters), iRegisterIndex := 308, iBitIndex := 10, xValue := stDumper.fbZQWarning[3].qxSignal);
FC_ModbusWriteBool(pRegisters := ADR(awModbusInputRegisters), iRegisterIndex := 308, iBitIndex := 11, xValue := stDumper.fbZQAlarm[3].qxSignal);
FC_ModbusWriteBool(pRegisters := ADR(awModbusInputRegisters), iRegisterIndex := 308, iBitIndex := 12, xValue := stDumper.fbZQWarning[4].qxSignal);
FC_ModbusWriteBool(pRegisters := ADR(awModbusInputRegisters), iRegisterIndex := 308, iBitIndex := 13, xValue := stDumper.fbZQAlarm[4].qxSignal);
FC_ModbusWriteBool(pRegisters := ADR(awModbusInputRegisters), iRegisterIndex := 308, iBitIndex := 14, xValue := stDumper.fbGS1.qxSignal);
FC_ModbusWriteBool(pRegisters := ADR(awModbusInputRegisters), iRegisterIndex := 308, iBitIndex := 15, xValue := stDumper.fbYS1.qxSignal);

FC_ModbusWriteBool(pRegisters := ADR(awModbusInputRegisters), iRegisterIndex := 309, iBitIndex := 0, xValue := stDumper.fbQR[1].qxSignal);
FC_ModbusWriteBool(pRegisters := ADR(awModbusInputRegisters), iRegisterIndex := 309, iBitIndex := 1, xValue := stDumper.fbQR[2].qxSignal);
FC_ModbusWriteBool(pRegisters := ADR(awModbusInputRegisters), iRegisterIndex := 309, iBitIndex := 2, xValue := stDumper.fbEndSwitchLeft.qxSignal);
FC_ModbusWriteBool(pRegisters := ADR(awModbusInputRegisters), iRegisterIndex := 309, iBitIndex := 3, xValue := stDumper.fbEndSwitchRight.qxSignal);
FC_ModbusWriteBool(pRegisters := ADR(awModbusInputRegisters), iRegisterIndex := 309, iBitIndex := 4, xValue := stDumper.MotorConveyor[1].fbStatorOverheat.qxSignal);
FC_ModbusWriteBool(pRegisters := ADR(awModbusInputRegisters), iRegisterIndex := 309, iBitIndex := 5, xValue := stDumper.MotorConveyor[2].fbStatorOverheat.qxSignal);
FC_ModbusWriteBool(pRegisters := ADR(awModbusInputRegisters), iRegisterIndex := 309, iBitIndex := 6, xValue := stDumper.MotorRotation[1].fbStatorOverheat.qxSignal);
FC_ModbusWriteBool(pRegisters := ADR(awModbusInputRegisters), iRegisterIndex := 309, iBitIndex := 7, xValue := stDumper.MotorRotation[2].fbStatorOverheat.qxSignal);

// Модуль DI6 (310-311): Отвалообразователь - Моторы и общие сигналы
FC_ModbusWriteBool(pRegisters := ADR(awModbusInputRegisters), iRegisterIndex := 310, iBitIndex := 0, xValue := stDumper.MotorConveyor[1].VFD.fbStateRdyToStart.qxSignal);
FC_ModbusWriteBool(pRegisters := ADR(awModbusInputRegisters), iRegisterIndex := 310, iBitIndex := 1, xValue := stDumper.MotorConveyor[1].VFD.fbStateIsWorking.qxSignal);
FC_ModbusWriteBool(pRegisters := ADR(awModbusInputRegisters), iRegisterIndex := 310, iBitIndex := 2, xValue := stDumper.MotorConveyor[1].VFD.fbStateFailure.qxSignal);
FC_ModbusWriteBool(pRegisters := ADR(awModbusInputRegisters), iRegisterIndex := 310, iBitIndex := 3, xValue := stDumper.MotorConveyor[1].fbStateQF.qxSignal);
FC_ModbusWriteBool(pRegisters := ADR(awModbusInputRegisters), iRegisterIndex := 310, iBitIndex := 4, xValue := stDumper.MotorConveyor[1].fbStateKM.qxSignal);
FC_ModbusWriteBool(pRegisters := ADR(awModbusInputRegisters), iRegisterIndex := 310, iBitIndex := 5, xValue := stDumper.MotorConveyor[2].VFD.fbStateRdyToStart.qxSignal);
FC_ModbusWriteBool(pRegisters := ADR(awModbusInputRegisters), iRegisterIndex := 310, iBitIndex := 6, xValue := stDumper.MotorConveyor[2].VFD.fbStateIsWorking.qxSignal);
FC_ModbusWriteBool(pRegisters := ADR(awModbusInputRegisters), iRegisterIndex := 310, iBitIndex := 7, xValue := stDumper.MotorConveyor[2].VFD.fbStateFailure.qxSignal);
FC_ModbusWriteBool(pRegisters := ADR(awModbusInputRegisters), iRegisterIndex := 310, iBitIndex := 8, xValue := stDumper.MotorConveyor[2].fbStateQF.qxSignal);
FC_ModbusWriteBool(pRegisters := ADR(awModbusInputRegisters), iRegisterIndex := 310, iBitIndex := 9, xValue := stDumper.MotorConveyor[2].fbStateKM.qxSignal);
FC_ModbusWriteBool(pRegisters := ADR(awModbusInputRegisters), iRegisterIndex := 310, iBitIndex := 10, xValue := stDumper.MotorRotation[1].VFD.fbStateRdyToStart.qxSignal);
FC_ModbusWriteBool(pRegisters := ADR(awModbusInputRegisters), iRegisterIndex := 310, iBitIndex := 11, xValue := stDumper.MotorRotation[1].VFD.fbStateIsWorking.qxSignal);
FC_ModbusWriteBool(pRegisters := ADR(awModbusInputRegisters), iRegisterIndex := 310, iBitIndex := 12, xValue := stDumper.MotorRotation[1].VFD.fbStateFailure.qxSignal);
FC_ModbusWriteBool(pRegisters := ADR(awModbusInputRegisters), iRegisterIndex := 310, iBitIndex := 13, xValue := stDumper.MotorRotation[1].fbRotationStatus.qxSignal);
FC_ModbusWriteBool(pRegisters := ADR(awModbusInputRegisters), iRegisterIndex := 310, iBitIndex := 14, xValue := stDumper.MotorRotation[1].fbStateQF.qxSignal);
FC_ModbusWriteBool(pRegisters := ADR(awModbusInputRegisters), iRegisterIndex := 310, iBitIndex := 15, xValue := stDumper.MotorRotation[1].fbStateKM.qxSignal);

FC_ModbusWriteBool(pRegisters := ADR(awModbusInputRegisters), iRegisterIndex := 311, iBitIndex := 0, xValue := stDumper.MotorRotation[2].VFD.fbStateRdyToStart.qxSignal);
FC_ModbusWriteBool(pRegisters := ADR(awModbusInputRegisters), iRegisterIndex := 311, iBitIndex := 1, xValue := stDumper.MotorRotation[2].VFD.fbStateIsWorking.qxSignal);
FC_ModbusWriteBool(pRegisters := ADR(awModbusInputRegisters), iRegisterIndex := 311, iBitIndex := 2, xValue := stDumper.MotorRotation[2].VFD.fbStateFailure.qxSignal);
FC_ModbusWriteBool(pRegisters := ADR(awModbusInputRegisters), iRegisterIndex := 311, iBitIndex := 3, xValue := stDumper.MotorRotation[2].fbRotationStatus.qxSignal);
FC_ModbusWriteBool(pRegisters := ADR(awModbusInputRegisters), iRegisterIndex := 311, iBitIndex := 4, xValue := stDumper.MotorRotation[2].fbStateQF.qxSignal);
FC_ModbusWriteBool(pRegisters := ADR(awModbusInputRegisters), iRegisterIndex := 311, iBitIndex := 5, xValue := stDumper.MotorRotation[2].fbStateKM.qxSignal);
FC_ModbusWriteBool(pRegisters := ADR(awModbusInputRegisters), iRegisterIndex := 311, iBitIndex := 6, xValue := stCommonSignals.fbRealyCurrentControl.qxSignal);
FC_ModbusWriteBool(pRegisters := ADR(awModbusInputRegisters), iRegisterIndex := 311, iBitIndex := 7, xValue := stCommonSignals.fb9QF1.qxSignal);
FC_ModbusWriteBool(pRegisters := ADR(awModbusInputRegisters), iRegisterIndex := 311, iBitIndex := 8, xValue := stCommonSignals.fb10QF1.qxSignal);
FC_ModbusWriteBool(pRegisters := ADR(awModbusInputRegisters), iRegisterIndex := 311, iBitIndex := 9, xValue := stCommonSignals.fb11QF1.qxSignal);
FC_ModbusWriteBool(pRegisters := ADR(awModbusInputRegisters), iRegisterIndex := 311, iBitIndex := 10, xValue := stCommonSignals.fbQF1.qxSignal);

// Модуль DI7 (312-313): Кнопки управления
FC_ModbusWriteBool(pRegisters := ADR(awModbusInputRegisters), iRegisterIndex := 312, iBitIndex := 0, xValue := stBunker[1].fbBtnStart.qxSignal);
FC_ModbusWriteBool(pRegisters := ADR(awModbusInputRegisters), iRegisterIndex := 312, iBitIndex := 1, xValue := stBunker[1].fbBtnStop.qxSignal);
FC_ModbusWriteBool(pRegisters := ADR(awModbusInputRegisters), iRegisterIndex := 312, iBitIndex := 2, xValue := stBunker[1].fbBtnEmergencyStop.qxSignal);
FC_ModbusWriteBool(pRegisters := ADR(awModbusInputRegisters), iRegisterIndex := 312, iBitIndex := 3, xValue := stBunker[2].fbBtnStart.qxSignal);
FC_ModbusWriteBool(pRegisters := ADR(awModbusInputRegisters), iRegisterIndex := 312, iBitIndex := 4, xValue := stBunker[2].fbBtnStop.qxSignal);
FC_ModbusWriteBool(pRegisters := ADR(awModbusInputRegisters), iRegisterIndex := 312, iBitIndex := 5, xValue := stBunker[2].fbBtnEmergencyStop.qxSignal);
FC_ModbusWriteBool(pRegisters := ADR(awModbusInputRegisters), iRegisterIndex := 312, iBitIndex := 6, xValue := stBunker[3].fbBtnStart.qxSignal);
FC_ModbusWriteBool(pRegisters := ADR(awModbusInputRegisters), iRegisterIndex := 312, iBitIndex := 7, xValue := stBunker[3].fbBtnStop.qxSignal);
FC_ModbusWriteBool(pRegisters := ADR(awModbusInputRegisters), iRegisterIndex := 312, iBitIndex := 8, xValue := stBunker[3].fbBtnEmergencyStop.qxSignal);
FC_ModbusWriteBool(pRegisters := ADR(awModbusInputRegisters), iRegisterIndex := 312, iBitIndex := 9, xValue := stConveyor.fbBtnStart.qxSignal);
FC_ModbusWriteBool(pRegisters := ADR(awModbusInputRegisters), iRegisterIndex := 312, iBitIndex := 10, xValue := stConveyor.fbBtnStop.qxSignal);
FC_ModbusWriteBool(pRegisters := ADR(awModbusInputRegisters), iRegisterIndex := 312, iBitIndex := 11, xValue := stConveyor.fbBtnEmergencyStop.qxSignal);
FC_ModbusWriteBool(pRegisters := ADR(awModbusInputRegisters), iRegisterIndex := 312, iBitIndex := 12, xValue := stDumper.fbBtnStart.qxSignal);
FC_ModbusWriteBool(pRegisters := ADR(awModbusInputRegisters), iRegisterIndex := 312, iBitIndex := 13, xValue := stDumper.fbBtnStop.qxSignal);
FC_ModbusWriteBool(pRegisters := ADR(awModbusInputRegisters), iRegisterIndex := 312, iBitIndex := 14, xValue := stDumper.fbBtnTurnLeft.qxSignal);
FC_ModbusWriteBool(pRegisters := ADR(awModbusInputRegisters), iRegisterIndex := 312, iBitIndex := 15, xValue := stDumper.fbBtnTurnRight.qxSignal);

FC_ModbusWriteBool(pRegisters := ADR(awModbusInputRegisters), iRegisterIndex := 313, iBitIndex := 0, xValue := stDumper.fbBtnEmergencyStop.qxSignal);
FC_ModbusWriteBool(pRegisters := ADR(awModbusInputRegisters), iRegisterIndex := 313, iBitIndex := 1, xValue := stCommonSignals.fbEmergencyStopBtn.qxSignal);
FC_ModbusWriteBool(pRegisters := ADR(awModbusInputRegisters), iRegisterIndex := 313, iBitIndex := 2, xValue := stCommonSignals.fbRemoteModeBtn.qxSignal);

// Модуль DI8 (314-315): Перегрев вибропитателей и выключатели
FC_ModbusWriteBool(pRegisters := ADR(awModbusInputRegisters), iRegisterIndex := 314, iBitIndex := 0, xValue := stBunker[1].MotorVibFeeder[1].fbStatorOverheat.qxSignal);
FC_ModbusWriteBool(pRegisters := ADR(awModbusInputRegisters), iRegisterIndex := 314, iBitIndex := 1, xValue := stBunker[1].MotorVibFeeder[2].fbStatorOverheat.qxSignal);
FC_ModbusWriteBool(pRegisters := ADR(awModbusInputRegisters), iRegisterIndex := 314, iBitIndex := 2, xValue := stBunker[2].MotorVibFeeder[1].fbStatorOverheat.qxSignal);
FC_ModbusWriteBool(pRegisters := ADR(awModbusInputRegisters), iRegisterIndex := 314, iBitIndex := 3, xValue := stBunker[2].MotorVibFeeder[2].fbStatorOverheat.qxSignal);
FC_ModbusWriteBool(pRegisters := ADR(awModbusInputRegisters), iRegisterIndex := 314, iBitIndex := 4, xValue := stBunker[3].MotorVibFeeder[1].fbStatorOverheat.qxSignal);
FC_ModbusWriteBool(pRegisters := ADR(awModbusInputRegisters), iRegisterIndex := 314, iBitIndex := 5, xValue := stBunker[3].MotorVibFeeder[2].fbStatorOverheat.qxSignal);
FC_ModbusWriteBool(pRegisters := ADR(awModbusInputRegisters), iRegisterIndex := 314, iBitIndex := 6, xValue := stConveyor.fbBreakerConveyor.qxSignal);
FC_ModbusWriteBool(pRegisters := ADR(awModbusInputRegisters), iRegisterIndex := 314, iBitIndex := 7, xValue := stDumper.fbBreakerConveyor.qxSignal);
FC_ModbusWriteBool(pRegisters := ADR(awModbusInputRegisters), iRegisterIndex := 314, iBitIndex := 8, xValue := stDumper.fbBreakerRotation.qxSignal);
